RoboDK station: NewNozzleTest.rdk

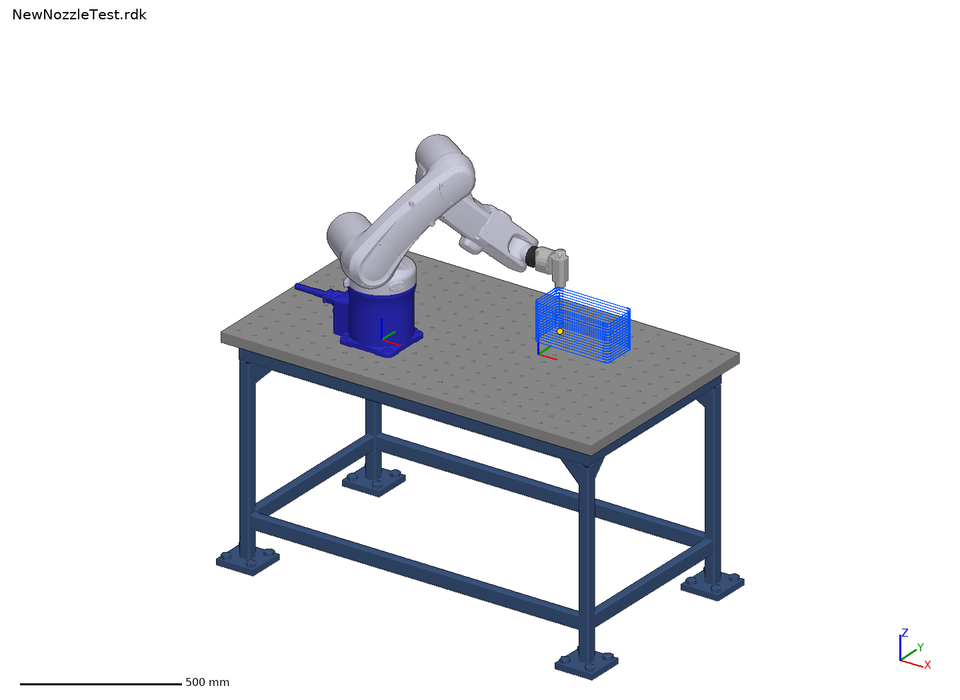
[picture v0: the station drawn from its stored meshes, robots at their saved joint values, targets as dots, program paths as lines]
Station NewNozzleTest (saved by RoboDK 5.5.4). Poses are relative to the parent item; angles as X-Y-Z fixed-axis rotations.
Station parameters (name, value as stored): TAGS, ['Additive Manufacturing', 'Additive manufacturing']
  - frame Denso VS-6577G-B Base at (0, 0, 0) mm
    - robot Denso VS-6577G-B: 6 axes, payload 7 kg, reach 854 mm, repeatability 0.03 mm, weight 36 kg
        modified DH rows (alpha deg, a mm, theta deg, d mm): 0, 0, 0, 335; -90, 75, -90, 0; 0, 365, -90, 0; -90, 90, 0, 405; 90, 0, 0, 0; -90, 0, 0, 80
        joint limits [-170, -100, -119, -190, -120, -360] to [170, 135, 169, 190, 120, 360]; home [0, 0, 90, 0, 0, 0]; saved at [-126.274, -49.631, -82.283, 63.884, 63.879, -41.926]
      - tool nozzle, TCP at (80, 0, 80) mm, rotated rx 0 ry 90 rz 0 deg, size 127 x 69.8 x 103.1 mm, geometry from nozzle.STEP
      - tool nozzle, TCP at (0, 0, 200) mm, size 127 x 76.2 x 113.3 mm, geometry from nozzle.STEP
    - object Table 1400x800x800mm at (-100, 160, 0) mm, size 1420 x 820 x 800 mm, geometry from Table-1400x800x800mm.sld
  - frame Reference at (454.66, 194.92, 0) mm
    - object Part at (0, 0, -20) mm, size 120 x 120 x 160 mm, geometry from part.sld
  - machining project Print3D settings: C:/Users/silverBlacK/OneDrive - University of Idaho/Research/RoboticsResearch/WallSection.gcode | rotZ(0) | rotX(0)*rotY(0) | rotZ(0)
  - program Print3D (17607 instructions, listed below)
  - Python program Extruder (listed below)
  - Python program SimulateFinalResult (listed below)
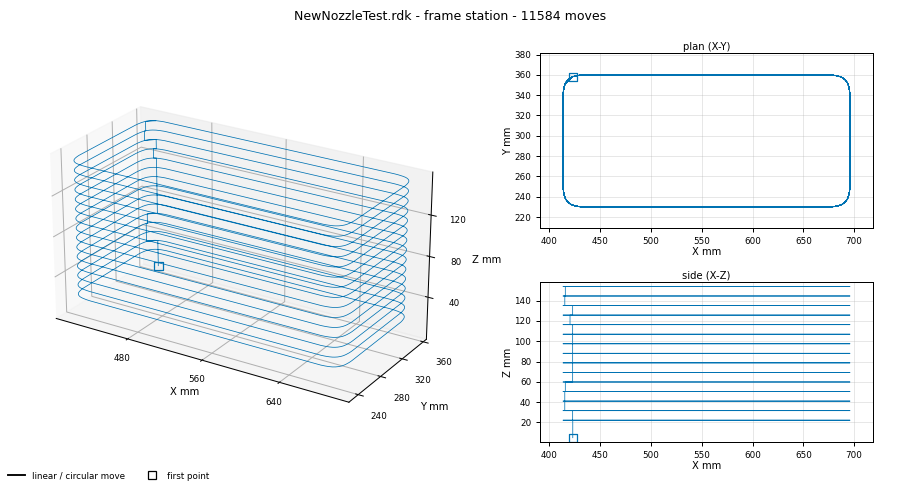
[picture p0: tool path of NewNozzleTest.rdk in frame station, 11584 of 11584 moves have a stored position in this frame; points joined in program order, loops and branches not executed]

--- program Print3D (robot Denso VS-6577G-B) ---
  Call M_RunCode(107)
  Call M_RunCode(104)
  Set speed (83.3 mm/s)
  Set speed (1000.0 mm/s)
  Set Ref.: Reference
  Set Tool: nozzle
  Show nozzle
  MoveJ 1 to (-31.64, 163.21, 5) mm, rotated rx -180 ry 0 rz 180 deg; joints [-126.294, -69.901, -72.383, 59.845, 68.77, -31.936]
  MoveL 2 to (-31.64, 163.21, 5) mm, rotated rx -180 ry 0 rz 180 deg; joints [-126.294, -69.901, -72.383, 59.845, 68.77, -31.936]
  Call Extruder(-1)
  MoveL 3 to (-31.64, 163.21, 5) mm, rotated rx -180 ry 0 rz 180 deg; joints [-126.294, -69.901, -72.383, 59.845, 68.77, -31.936]
  Call M_RunCode(109)
  Call M_RunCode(82)
  Call Extruder(0.00000)
  Set speed (130.0 mm/s)
  MoveL 4 to (-31.64, 163.21, 22.22) mm, rotated rx -180 ry 0 rz -180 deg; joints [-126.294, -67.456, -73.96, 60.14, 68.336, -32.743]
  Call Extruder(-2.00000)
  Set speed (40.0 mm/s)
  MoveL 5 to (-31.64, 163.21, 22.22) mm, rotated rx -180 ry 0 rz -180 deg; joints [-126.294, -67.456, -73.96, 60.14, 68.336, -32.743]
  Call Extruder(0.00000)
  Set speed (130.0 mm/s)
  MoveL 6 to (-31.64, 163.21, 22.22) mm, rotated rx -180 ry 0 rz -180 deg; joints [-126.294, -67.456, -73.96, 60.14, 68.336, -32.743]
  Call Extruder(2.00000)
  Set speed (40.0 mm/s)
  MoveL 7 to (-31.64, 163.21, 22.22) mm, rotated rx -180 ry 0 rz -180 deg; joints [-126.294, -67.456, -73.96, 60.14, 68.336, -32.743]
  Set speed (30.0 mm/s)
  MoveL 8 to (-31.64, 163.21, 22.22) mm, rotated rx -180 ry 0 rz -180 deg; joints [-126.294, -67.456, -73.96, 60.14, 68.336, -32.743]
  Call Extruder(2.38024)
  MoveL 9 to (-31.93, 163.09, 22.23) mm, rotated rx 180 ry 0 rz -180 deg; joints [-126.273, -67.437, -74.013, 60.147, 68.364, -32.718]
  MoveL 10 to (-31.93, 163.09, 22.23) mm, rotated rx 180 ry 0 rz -180 deg; joints [-126.273, -67.437, -74.013, 60.147, 68.364, -32.718]
  Call Extruder(2.76227)
  MoveL 11 to (-32.22, 162.97, 22.23) mm, rotated rx 180 ry 0 rz 180 deg; joints [-126.252, -67.418, -74.067, 60.155, 68.393, -32.692]
  MoveL 12 to (-32.22, 162.97, 22.23) mm, rotated rx 180 ry 0 rz 180 deg; joints [-126.252, -67.418, -74.067, 60.155, 68.393, -32.692]
  Call Extruder(3.11872)
  MoveL 13 to (-32.49, 162.85, 22.23) mm, rotated rx -180 ry 0 rz 180 deg; joints [-126.233, -67.401, -74.116, 60.161, 68.419, -32.669]
  MoveL 14 to (-32.49, 162.85, 22.23) mm, rotated rx -180 ry 0 rz 180 deg; joints [-126.233, -67.401, -74.116, 60.161, 68.419, -32.669]
  Call Extruder(3.44932)
  MoveL 15 to (-32.74, 162.74, 22.23) mm, rotated rx 180 ry 0 rz -180 deg; joints [-126.215, -67.385, -74.162, 60.167, 68.444, -32.647]
  MoveL 16 to (-32.74, 162.74, 22.23) mm, rotated rx 180 ry 0 rz -180 deg; joints [-126.215, -67.385, -74.162, 60.167, 68.444, -32.647]
  Call Extruder(3.78134)
  MoveL 17 to (-32.99, 162.64, 22.22) mm, rotated rx -180 ry 0 rz 180 deg; joints [-126.197, -67.369, -74.208, 60.173, 68.468, -32.625]
  MoveL 18 to (-32.99, 162.64, 22.22) mm, rotated rx -180 ry 0 rz 180 deg; joints [-126.197, -67.369, -74.208, 60.173, 68.468, -32.625]
  Call Extruder(4.21321)
  MoveL 19 to (-33.29, 162.46, 22.23) mm, rotated rx -180 ry 0 rz 180 deg; joints [-126.179, -67.347, -74.271, 60.176, 68.499, -32.593]
  MoveL 20 to (-33.29, 162.46, 22.23) mm, rotated rx -180 ry 0 rz 180 deg; joints [-126.179, -67.347, -74.271, 60.176, 68.499, -32.593]
  Call Extruder(4.64692)
  MoveL 21 to (-33.6, 162.29, 22.22) mm, rotated rx 180 ry 0 rz -180 deg; joints [-126.16, -67.325, -74.334, 60.178, 68.529, -32.561]
  MoveL 22 to (-33.6, 162.29, 22.22) mm, rotated rx 180 ry 0 rz -180 deg; joints [-126.16, -67.325, -74.334, 60.178, 68.529, -32.561]
  Call Extruder(5.08247)
  MoveL 23 to (-33.9, 162.11, 22.23) mm, rotated rx 180 ry 0 rz 180 deg; joints [-126.142, -67.303, -74.397, 60.181, 68.559, -32.529]
  MoveL 24 to (-33.9, 162.11, 22.23) mm, rotated rx 180 ry 0 rz 180 deg; joints [-126.142, -67.303, -74.397, 60.181, 68.559, -32.529]
  Call Extruder(5.51986)
  MoveL 25 to (-34.21, 161.94, 22.23) mm, rotated rx 180 ry 0 rz 180 deg; joints [-126.123, -67.281, -74.46, 60.184, 68.589, -32.497]
  MoveL 26 to (-34.21, 161.94, 22.23) mm, rotated rx 180 ry 0 rz 180 deg; joints [-126.123, -67.281, -74.46, 60.184, 68.589, -32.497]
  Call Extruder(5.89660)
  MoveL 27 to (-34.45, 161.76, 22.23) mm, rotated rx 180 ry 0 rz 180 deg; joints [-126.111, -67.261, -74.516, 60.182, 68.614, -32.467]
  MoveL 28 to (-34.45, 161.76, 22.23) mm, rotated rx 180 ry 0 rz 180 deg; joints [-126.111, -67.261, -74.516, 60.182, 68.614, -32.467]
  Call Extruder(6.59657)
  MoveL 29 to (-34.9, 161.43, 22.23) mm, rotated rx -180 ry 0 rz 180 deg; joints [-126.089, -67.225, -74.62, 60.18, 68.66, -32.411]
  MoveL 30 to (-34.9, 161.43, 22.23) mm, rotated rx -180 ry 0 rz 180 deg; joints [-126.089, -67.225, -74.62, 60.18, 68.66, -32.411]
  Call Extruder(7.29934)
  MoveL 31 to (-35.35, 161.1, 22.22) mm, rotated rx 180 ry 0 rz 180 deg; joints [-126.067, -67.189, -74.723, 60.177, 68.705, -32.355]
  Call Extruder(9.03811)
  MoveL 32 to (-36.39, 160.19, 22.22) mm, rotated rx 180 ry 0 rz 180 deg; joints [-126.027, -67.098, -74.986, 60.155, 68.812, -32.208]
  Call Extruder(10.77694)
  MoveL 33 to (-37.3, 159.15, 22.22) mm, rotated rx 180 ry 0 rz -180 deg; joints [-126.011, -67.006, -75.254, 60.111, 68.908, -32.051]
  Call Extruder(11.12832)
  MoveL 34 to (-37.47, 158.93, 22.22) mm, rotated rx -180 ry 0 rz 180 deg; joints [-126.011, -66.987, -75.308, 60.099, 68.926, -32.018]
  MoveL 35 to (-37.47, 158.93, 22.22) mm, rotated rx -180 ry 0 rz 180 deg; joints [-126.011, -66.987, -75.308, 60.099, 68.926, -32.018]
  Call Extruder(11.82828)
  MoveL 36 to (-37.79, 158.48, 22.22) mm, rotated rx 180 ry 0 rz 180 deg; joints [-126.011, -66.95, -75.416, 60.076, 68.961, -31.952]
  MoveL 37 to (-37.79, 158.48, 22.22) mm, rotated rx 180 ry 0 rz 180 deg; joints [-126.011, -66.95, -75.416, 60.076, 68.961, -31.952]
  Call Extruder(12.52544)
  MoveL 38 to (-38.12, 158.03, 22.23) mm, rotated rx 180 ry 0 rz 180 deg; joints [-126.011, -66.913, -75.524, 60.052, 68.996, -31.886]
  MoveL 39 to (-38.12, 158.03, 22.23) mm, rotated rx 180 ry 0 rz 180 deg; joints [-126.011, -66.913, -75.524, 60.052, 68.996, -31.886]
  Call Extruder(12.77229)
  MoveL 40 to (-38.22, 157.85, 22.23) mm, rotated rx 180 ry 0 rz -180 deg; joints [-126.013, -66.9, -75.562, 60.041, 69.008, -31.862]
  MoveL 41 to (-38.22, 157.85, 22.23) mm, rotated rx 180 ry 0 rz -180 deg; joints [-126.013, -66.9, -75.562, 60.041, 69.008, -31.862]
  Call Extruder(13.20785)
  MoveL 42 to (-38.4, 157.55, 22.22) mm, rotated rx -180 ry 0 rz -180 deg; joints [-126.018, -66.876, -75.63, 60.022, 69.027, -31.82]
  MoveL 43 to (-38.4, 157.55, 22.22) mm, rotated rx -180 ry 0 rz -180 deg; joints [-126.018, -66.876, -75.63, 60.022, 69.027, -31.82]
  Call Extruder(13.64157)
  MoveL 44 to (-38.57, 157.25, 22.22) mm, rotated rx 180 ry 0 rz -180 deg; joints [-126.023, -66.853, -75.697, 60.003, 69.047, -31.777]
  MoveL 45 to (-38.57, 157.25, 22.22) mm, rotated rx 180 ry 0 rz -180 deg; joints [-126.023, -66.853, -75.697, 60.003, 69.047, -31.777]
  Call Extruder(14.07344)
  MoveL 46 to (-38.75, 156.94, 22.22) mm, rotated rx -180 ry 0 rz -180 deg; joints [-126.028, -66.83, -75.765, 59.984, 69.066, -31.734]
  MoveL 47 to (-38.75, 156.94, 22.22) mm, rotated rx -180 ry 0 rz -180 deg; joints [-126.028, -66.83, -75.765, 59.984, 69.066, -31.734]
  Call Extruder(14.45383)
  MoveL 48 to (-38.89, 156.67, 22.22) mm, rotated rx -180 ry 0 rz -180 deg; joints [-126.034, -66.81, -75.824, 59.965, 69.083, -31.696]
  MoveL 49 to (-38.89, 156.67, 22.22) mm, rotated rx -180 ry 0 rz -180 deg; joints [-126.034, -66.81, -75.824, 59.965, 69.083, -31.696]
  Call Extruder(14.78446)
  MoveL 50 to (-39, 156.42, 22.22) mm, rotated rx -180 ry 0 rz -180 deg; joints [-126.042, -66.793, -75.875, 59.947, 69.095, -31.662]
  MoveL 51 to (-39, 156.42, 22.22) mm, rotated rx -180 ry 0 rz -180 deg; joints [-126.042, -66.793, -75.875, 59.947, 69.095, -31.662]
  Call Extruder(15.11366)
  MoveL 52 to (-39.1, 156.17, 22.23) mm, rotated rx -180 ry 0 rz 180 deg; joints [-126.05, -66.775, -75.926, 59.929, 69.108, -31.629]
  MoveL 53 to (-39.1, 156.17, 22.23) mm, rotated rx -180 ry 0 rz 180 deg; joints [-126.05, -66.775, -75.926, 59.929, 69.108, -31.629]
  Call Extruder(15.49565)
  MoveL 54 to (-39.23, 155.87, 22.22) mm, rotated rx -180 ry 0 rz -180 deg; joints [-126.06, -66.755, -75.985, 59.907, 69.122, -31.589]
  MoveL 55 to (-39.23, 155.87, 22.22) mm, rotated rx -180 ry 0 rz -180 deg; joints [-126.06, -66.755, -75.985, 59.907, 69.122, -31.589]
  Call Extruder(15.87585)
  MoveL 56 to (-39.35, 155.58, 22.22) mm, rotated rx -180 ry 0 rz 180 deg; joints [-126.07, -66.735, -76.044, 59.885, 69.137, -31.55]
  MoveL 57 to (-39.35, 155.58, 22.22) mm, rotated rx -180 ry 0 rz 180 deg; joints [-126.07, -66.735, -76.044, 59.885, 69.137, -31.55]
  Call Extruder(16.18353)
  MoveL 58 to (-39.44, 155.34, 22.22) mm, rotated rx 180 ry 0 rz -180 deg; joints [-126.079, -66.719, -76.092, 59.866, 69.148, -31.518]
  MoveL 59 to (-39.44, 155.34, 22.22) mm, rotated rx 180 ry 0 rz -180 deg; joints [-126.079, -66.719, -76.092, 59.866, 69.148, -31.518]
  Call Extruder(16.41988)
  MoveL 60 to (-39.5, 155.15, 22.22) mm, rotated rx -180 ry 0 rz 180 deg; joints [-126.087, -66.706, -76.128, 59.851, 69.156, -31.493]
  MoveL 61 to (-39.5, 155.15, 22.22) mm, rotated rx -180 ry 0 rz 180 deg; joints [-126.087, -66.706, -76.128, 59.851, 69.156, -31.493]
  Call Extruder(16.65518)
  MoveL 62 to (-39.56, 154.97, 22.23) mm, rotated rx 180 ry 0 rz -180 deg; joints [-126.095, -66.694, -76.164, 59.836, 69.163, -31.468]
  MoveL 63 to (-39.56, 154.97, 22.23) mm, rotated rx 180 ry 0 rz -180 deg; joints [-126.095, -66.694, -76.164, 59.836, 69.163, -31.468]
  Call Extruder(16.88943)
  MoveL 64 to (-39.62, 154.78, 22.22) mm, rotated rx -180 ry 0 rz -180 deg; joints [-126.103, -66.682, -76.201, 59.82, 69.171, -31.444]
  MoveL 65 to (-39.62, 154.78, 22.22) mm, rotated rx -180 ry 0 rz -180 deg; joints [-126.103, -66.682, -76.201, 59.82, 69.171, -31.444]
  Call Extruder(17.12262)
  MoveL 66 to (-39.68, 154.59, 22.22) mm, rotated rx 180 ry 0 rz 180 deg; joints [-126.111, -66.669, -76.237, 59.805, 69.179, -31.419]
  MoveL 67 to (-39.68, 154.59, 22.22) mm, rotated rx 180 ry 0 rz 180 deg; joints [-126.111, -66.669, -76.237, 59.805, 69.179, -31.419]
  Call Extruder(17.37548)
  MoveL 68 to (-39.75, 154.38, 22.22) mm, rotated rx 180 ry 0 rz 180 deg; joints [-126.12, -66.656, -76.276, 59.788, 69.187, -31.392]
  MoveL 69 to (-39.75, 154.38, 22.22) mm, rotated rx 180 ry 0 rz 180 deg; joints [-126.12, -66.656, -76.276, 59.788, 69.187, -31.392]
  Call Extruder(17.64775)
  MoveL 70 to (-39.81, 154.16, 22.23) mm, rotated rx 180 ry 0 rz 180 deg; joints [-126.131, -66.642, -76.318, 59.77, 69.196, -31.363]
  MoveL 71 to (-39.81, 154.16, 22.23) mm, rotated rx 180 ry 0 rz 180 deg; joints [-126.131, -66.642, -76.318, 59.77, 69.196, -31.363]
  Call Extruder(17.91868)
  MoveL 72 to (-39.88, 153.94, 22.23) mm, rotated rx -180 ry 0 rz 180 deg; joints [-126.141, -66.627, -76.361, 59.751, 69.205, -31.334]
  MoveL 73 to (-39.88, 153.94, 22.23) mm, rotated rx -180 ry 0 rz 180 deg; joints [-126.141, -66.627, -76.361, 59.751, 69.205, -31.334]
  Call Extruder(18.18828)
  MoveL 74 to (-39.95, 153.71, 22.23) mm, rotated rx 180 ry 0 rz -180 deg; joints [-126.151, -66.613, -76.403, 59.733, 69.213, -31.305]
  MoveL 75 to (-39.95, 153.71, 22.23) mm, rotated rx 180 ry 0 rz -180 deg; joints [-126.151, -66.613, -76.403, 59.733, 69.213, -31.305]
  Call Extruder(18.45654)
  MoveL 76 to (-40.02, 153.49, 22.22) mm, rotated rx -180 ry 0 rz 180 deg; joints [-126.161, -66.599, -76.445, 59.714, 69.222, -31.275]
  MoveL 77 to (-40.02, 153.49, 22.22) mm, rotated rx -180 ry 0 rz 180 deg; joints [-126.161, -66.599, -76.445, 59.714, 69.222, -31.275]
  Call Extruder(18.69554)
  MoveL 78 to (-40.06, 153.28, 22.23) mm, rotated rx 180 ry 0 rz 180 deg; joints [-126.173, -66.586, -76.482, 59.696, 69.228, -31.249]
  MoveL 79 to (-40.06, 153.28, 22.23) mm, rotated rx 180 ry 0 rz 180 deg; joints [-126.173, -66.586, -76.482, 59.696, 69.228, -31.249]
  Call Extruder(18.93348)
  MoveL 80 to (-40.11, 153.08, 22.23) mm, rotated rx 180 ry 0 rz 180 deg; joints [-126.184, -66.574, -76.518, 59.678, 69.235, -31.223]
  MoveL 81 to (-40.11, 153.08, 22.23) mm, rotated rx 180 ry 0 rz 180 deg; joints [-126.184, -66.574, -76.518, 59.678, 69.235, -31.223]
  Call Extruder(19.17035)
  MoveL 82 to (-40.15, 152.88, 22.22) mm, rotated rx 180 ry 0 rz 180 deg; joints [-126.195, -66.561, -76.555, 59.66, 69.241, -31.197]
  MoveL 83 to (-40.15, 152.88, 22.22) mm, rotated rx 180 ry 0 rz 180 deg; joints [-126.195, -66.561, -76.555, 59.66, 69.241, -31.197]
  Call Extruder(19.40615)
  MoveL 84 to (-40.2, 152.67, 22.22) mm, rotated rx -180 ry 0 rz 180 deg; joints [-126.206, -66.549, -76.592, 59.641, 69.248, -31.171]
  MoveL 85 to (-40.2, 152.67, 22.22) mm, rotated rx -180 ry 0 rz 180 deg; joints [-126.206, -66.549, -76.592, 59.641, 69.248, -31.171]
  Call Extruder(19.66605)
  MoveL 86 to (-40.24, 152.45, 22.23) mm, rotated rx 180 ry 0 rz 180 deg; joints [-126.219, -66.535, -76.632, 59.621, 69.255, -31.143]
  MoveL 87 to (-40.24, 152.45, 22.23) mm, rotated rx 180 ry 0 rz 180 deg; joints [-126.219, -66.535, -76.632, 59.621, 69.255, -31.143]
  Call Extruder(19.94972)
  MoveL 88 to (-40.29, 152.2, 22.22) mm, rotated rx 180 ry 0 rz -180 deg; joints [-126.233, -66.521, -76.676, 59.598, 69.262, -31.111]
  MoveL 89 to (-40.29, 152.2, 22.22) mm, rotated rx 180 ry 0 rz -180 deg; joints [-126.233, -66.521, -76.676, 59.598, 69.262, -31.111]
  Call Extruder(20.23193)
  MoveL 90 to (-40.34, 151.95, 22.22) mm, rotated rx -180 ry 0 rz 180 deg; joints [-126.248, -66.506, -76.72, 59.576, 69.269, -31.079]
  MoveL 91 to (-40.34, 151.95, 22.22) mm, rotated rx -180 ry 0 rz 180 deg; joints [-126.248, -66.506, -76.72, 59.576, 69.269, -31.079]
  Call Extruder(20.51271)
  MoveL 92 to (-40.39, 151.7, 22.23) mm, rotated rx 180 ry 0 rz 180 deg; joints [-126.262, -66.491, -76.764, 59.553, 69.277, -31.048]
  MoveL 93 to (-40.39, 151.7, 22.23) mm, rotated rx 180 ry 0 rz 180 deg; joints [-126.262, -66.491, -76.764, 59.553, 69.277, -31.048]
  Call Extruder(20.79205)
  MoveL 94 to (-40.44, 151.45, 22.22) mm, rotated rx -180 ry 0 rz 180 deg; joints [-126.276, -66.476, -76.808, 59.53, 69.284, -31.016]
  MoveL 95 to (-40.44, 151.45, 22.22) mm, rotated rx -180 ry 0 rz 180 deg; joints [-126.276, -66.476, -76.808, 59.53, 69.284, -31.016]
  Call Extruder(21.06994)
  MoveL 96 to (-40.49, 151.2, 22.23) mm, rotated rx 180 ry 0 rz 180 deg; joints [-126.291, -66.461, -76.852, 59.508, 69.292, -30.985]
  MoveL 97 to (-40.49, 151.2, 22.23) mm, rotated rx 180 ry 0 rz 180 deg; joints [-126.291, -66.461, -76.852, 59.508, 69.292, -30.985]
  Call Extruder(21.34639)
  MoveL 98 to (-40.54, 150.95, 22.22) mm, rotated rx -180 ry 0 rz -180 deg; joints [-126.305, -66.447, -76.896, 59.485, 69.299, -30.953]
  MoveL 99 to (-40.54, 150.95, 22.22) mm, rotated rx -180 ry 0 rz -180 deg; joints [-126.305, -66.447, -76.896, 59.485, 69.299, -30.953]
  Call Extruder(21.65140)
  MoveL 100 to (-40.59, 150.67, 22.22) mm, rotated rx 180 ry 0 rz 180 deg; joints [-126.322, -66.43, -76.944, 59.46, 69.307, -30.919]
  MoveL 101 to (-40.59, 150.67, 22.22) mm, rotated rx 180 ry 0 rz 180 deg; joints [-126.322, -66.43, -76.944, 59.46, 69.307, -30.919]
  Call Extruder(21.98479)
  MoveL 102 to (-40.64, 150.37, 22.22) mm, rotated rx -180 ry 0 rz 180 deg; joints [-126.341, -66.413, -76.996, 59.431, 69.315, -30.88]
  MoveL 103 to (-40.64, 150.37, 22.22) mm, rotated rx -180 ry 0 rz 180 deg; joints [-126.341, -66.413, -76.996, 59.431, 69.315, -30.88]
  Call Extruder(22.31647)
  MoveL 104 to (-40.69, 150.06, 22.23) mm, rotated rx -180 ry 0 rz 180 deg; joints [-126.36, -66.395, -77.049, 59.402, 69.322, -30.842]
  MoveL 105 to (-40.69, 150.06, 22.23) mm, rotated rx -180 ry 0 rz 180 deg; joints [-126.36, -66.395, -77.049, 59.402, 69.322, -30.842]
  Call Extruder(22.64643)
  MoveL 106 to (-40.74, 149.76, 22.22) mm, rotated rx -180 ry 0 rz -180 deg; joints [-126.379, -66.378, -77.101, 59.373, 69.33, -30.804]
  MoveL 107 to (-40.74, 149.76, 22.22) mm, rotated rx -180 ry 0 rz -180 deg; joints [-126.379, -66.378, -77.101, 59.373, 69.33, -30.804]
  Call Extruder(22.97467)
  MoveL 108 to (-40.78, 149.45, 22.22) mm, rotated rx -180 ry 0 rz -180 deg; joints [-126.398, -66.36, -77.153, 59.344, 69.338, -30.766]
  MoveL 109 to (-40.78, 149.45, 22.22) mm, rotated rx -180 ry 0 rz -180 deg; joints [-126.398, -66.36, -77.153, 59.344, 69.338, -30.766]
  Call Extruder(23.30119)
  MoveL 110 to (-40.83, 149.14, 22.22) mm, rotated rx 180 ry 0 rz -180 deg; joints [-126.417, -66.343, -77.206, 59.316, 69.346, -30.728]
  MoveL 111 to (-40.83, 149.14, 22.22) mm, rotated rx 180 ry 0 rz -180 deg; joints [-126.417, -66.343, -77.206, 59.316, 69.346, -30.728]
  Call Extruder(23.66827)
  MoveL 112 to (-40.88, 148.8, 22.22) mm, rotated rx 180 ry 0 rz -180 deg; joints [-126.439, -66.323, -77.264, 59.282, 69.355, -30.685]
  MoveL 113 to (-40.88, 148.8, 22.22) mm, rotated rx 180 ry 0 rz -180 deg; joints [-126.439, -66.323, -77.264, 59.282, 69.355, -30.685]
  Call Extruder(24.07571)
  MoveL 114 to (-40.92, 148.41, 22.22) mm, rotated rx -180 ry 0 rz 180 deg; joints [-126.465, -66.301, -77.328, 59.245, 69.363, -30.637]
  MoveL 115 to (-40.92, 148.41, 22.22) mm, rotated rx -180 ry 0 rz 180 deg; joints [-126.465, -66.301, -77.328, 59.245, 69.363, -30.637]
  Call Extruder(24.48110)
  MoveL 116 to (-40.97, 148.02, 22.22) mm, rotated rx -180 ry 0 rz -180 deg; joints [-126.491, -66.28, -77.393, 59.207, 69.372, -30.589]
  MoveL 117 to (-40.97, 148.02, 22.22) mm, rotated rx -180 ry 0 rz -180 deg; joints [-126.491, -66.28, -77.393, 59.207, 69.372, -30.589]
  Call Extruder(24.88445)
  MoveL 118 to (-41.02, 147.63, 22.23) mm, rotated rx 180 ry 0 rz -180 deg; joints [-126.517, -66.259, -77.457, 59.169, 69.381, -30.542]
  MoveL 119 to (-41.02, 147.63, 22.23) mm, rotated rx 180 ry 0 rz -180 deg; joints [-126.517, -66.259, -77.457, 59.169, 69.381, -30.542]
  Call Extruder(25.28574)
  MoveL 120 to (-41.06, 147.25, 22.22) mm, rotated rx -180 ry 0 rz 180 deg; joints [-126.543, -66.237, -77.521, 59.131, 69.389, -30.494]
  MoveL 121 to (-41.06, 147.25, 22.22) mm, rotated rx -180 ry 0 rz 180 deg; joints [-126.543, -66.237, -77.521, 59.131, 69.389, -30.494]
  Call Extruder(25.89062)
  MoveL 122 to (-41.11, 146.66, 22.23) mm, rotated rx -180 ry 0 rz 180 deg; joints [-126.585, -66.206, -77.616, 59.072, 69.401, -30.422]
  MoveL 123 to (-41.11, 146.66, 22.23) mm, rotated rx -180 ry 0 rz 180 deg; joints [-126.585, -66.206, -77.616, 59.072, 69.401, -30.422]
  Call Extruder(26.49235)
  MoveL 124 to (-41.15, 146.07, 22.23) mm, rotated rx 180 ry 0 rz -180 deg; joints [-126.628, -66.174, -77.711, 59.013, 69.412, -30.35]
  MoveL 125 to (-41.15, 146.07, 22.23) mm, rotated rx 180 ry 0 rz -180 deg; joints [-126.628, -66.174, -77.711, 59.013, 69.412, -30.35]
  Call Extruder(27.09093)
  MoveL 126 to (-41.2, 145.48, 22.23) mm, rotated rx -180 ry 0 rz 180 deg; joints [-126.67, -66.143, -77.806, 58.953, 69.423, -30.279]
  MoveL 127 to (-41.2, 145.48, 22.23) mm, rotated rx -180 ry 0 rz 180 deg; joints [-126.67, -66.143, -77.806, 58.953, 69.423, -30.279]
  Call Extruder(28.26271)
  MoveL 128 to (-41.25, 144.32, 22.23) mm, rotated rx 180 ry 0 rz 180 deg; joints [-126.759, -66.083, -77.987, 58.832, 69.441, -30.139]
  MoveL 129 to (-41.25, 144.32, 22.23) mm, rotated rx 180 ry 0 rz 180 deg; joints [-126.759, -66.083, -77.987, 58.832, 69.441, -30.139]
  Call Extruder(29.72057)
  MoveL 130 to (-41.29, 142.86, 22.23) mm, rotated rx 180 ry 0 rz 180 deg; joints [-126.873, -66.009, -78.211, 58.679, 69.462, -29.965]
  Call Extruder(115.61408)
  MoveL 131 to (-41.29, 57.14, 22.22) mm, rotated rx 180 ry 0 rz 180 deg; joints [-135.148, -62.641, -89.71, 48.318, 70.793, -20.278]
  Call Extruder(116.48916)
  MoveL 132 to (-41.27, 56.26, 22.23) mm, rotated rx 180 ry 0 rz 180 deg; joints [-135.25, -62.616, -89.811, 48.198, 70.808, -20.185]
  MoveL 133 to (-41.27, 56.26, 22.23) mm, rotated rx 180 ry 0 rz 180 deg; joints [-135.25, -62.616, -89.811, 48.198, 70.808, -20.185]
  Call Extruder(117.66094)
  MoveL 134 to (-41.23, 55.1, 22.22) mm, rotated rx -180 ry 0 rz 180 deg; joints [-135.387, -62.583, -89.942, 48.035, 70.826, -20.063]
  MoveL 135 to (-41.23, 55.1, 22.22) mm, rotated rx -180 ry 0 rz 180 deg; joints [-135.387, -62.583, -89.942, 48.035, 70.826, -20.063]
  Call Extruder(118.54904)
  MoveL 136 to (-41.18, 54.23, 22.23) mm, rotated rx 180 ry 0 rz 180 deg; joints [-135.493, -62.559, -90.039, 47.911, 70.839, -19.971]
  MoveL 137 to (-41.18, 54.23, 22.23) mm, rotated rx 180 ry 0 rz 180 deg; joints [-135.493, -62.559, -90.039, 47.911, 70.839, -19.971]
  Call Extruder(119.15077)
  MoveL 138 to (-41.13, 53.64, 22.23) mm, rotated rx 180 ry 0 rz 180 deg; joints [-135.566, -62.543, -90.102, 47.826, 70.846, -19.909]
  MoveL 139 to (-41.13, 53.64, 22.23) mm, rotated rx 180 ry 0 rz 180 deg; joints [-135.566, -62.543, -90.102, 47.826, 70.846, -19.909]
  Call Extruder(119.75565)
  MoveL 140 to (-41.09, 53.05, 22.22) mm, rotated rx -180 ry 0 rz -180 deg; joints [-135.64, -62.528, -90.165, 47.741, 70.853, -19.848]
  MoveL 141 to (-41.09, 53.05, 22.22) mm, rotated rx -180 ry 0 rz -180 deg; joints [-135.64, -62.528, -90.165, 47.741, 70.853, -19.848]
  Call Extruder(120.26021)
  MoveL 142 to (-41.04, 52.56, 22.23) mm, rotated rx 180 ry 0 rz 180 deg; joints [-135.701, -62.515, -90.217, 47.67, 70.858, -19.798]
  MoveL 143 to (-41.04, 52.56, 22.23) mm, rotated rx 180 ry 0 rz 180 deg; joints [-135.701, -62.515, -90.217, 47.67, 70.858, -19.798]
  Call Extruder(120.66355)
  MoveL 144 to (-40.99, 52.17, 22.23) mm, rotated rx -180 ry 0 rz 180 deg; joints [-135.751, -62.505, -90.256, 47.612, 70.862, -19.758]
  MoveL 145 to (-40.99, 52.17, 22.23) mm, rotated rx -180 ry 0 rz 180 deg; joints [-135.751, -62.505, -90.256, 47.612, 70.862, -19.758]
  Call Extruder(121.06894)
  MoveL 146 to (-40.95, 51.78, 22.23) mm, rotated rx 180 ry 0 rz 180 deg; joints [-135.801, -62.496, -90.296, 47.554, 70.865, -19.718]
  MoveL 147 to (-40.95, 51.78, 22.23) mm, rotated rx 180 ry 0 rz 180 deg; joints [-135.801, -62.496, -90.296, 47.554, 70.865, -19.718]
  Call Extruder(121.47639)
  MoveL 148 to (-40.9, 51.4, 22.23) mm, rotated rx 180 ry 0 rz -180 deg; joints [-135.852, -62.486, -90.335, 47.497, 70.868, -19.679]
  MoveL 149 to (-40.9, 51.4, 22.23) mm, rotated rx 180 ry 0 rz -180 deg; joints [-135.852, -62.486, -90.335, 47.497, 70.868, -19.679]
  Call Extruder(121.88588)
  MoveL 150 to (-40.86, 51.01, 22.23) mm, rotated rx 180 ry 0 rz 180 deg; joints [-135.902, -62.476, -90.375, 47.439, 70.871, -19.639]
  MoveL 151 to (-40.86, 51.01, 22.23) mm, rotated rx 180 ry 0 rz 180 deg; joints [-135.902, -62.476, -90.375, 47.439, 70.871, -19.639]
  Call Extruder(122.21240)
  MoveL 152 to (-40.81, 50.7, 22.23) mm, rotated rx 180 ry 0 rz -180 deg; joints [-135.943, -62.469, -90.404, 47.392, 70.873, -19.608]
  MoveL 153 to (-40.81, 50.7, 22.23) mm, rotated rx 180 ry 0 rz -180 deg; joints [-135.943, -62.469, -90.404, 47.392, 70.873, -19.608]
  Call Extruder(122.54064)
  MoveL 154 to (-40.76, 50.4, 22.22) mm, rotated rx 180 ry 0 rz -180 deg; joints [-135.984, -62.462, -90.434, 47.346, 70.874, -19.577]
  MoveL 155 to (-40.76, 50.4, 22.22) mm, rotated rx 180 ry 0 rz -180 deg; joints [-135.984, -62.462, -90.434, 47.346, 70.874, -19.577]
  Call Extruder(122.87060)
  MoveL 156 to (-40.71, 50.09, 22.23) mm, rotated rx 180 ry 0 rz 180 deg; joints [-136.025, -62.455, -90.463, 47.299, 70.875, -19.547]
  MoveL 157 to (-40.71, 50.09, 22.23) mm, rotated rx 180 ry 0 rz 180 deg; joints [-136.025, -62.455, -90.463, 47.299, 70.875, -19.547]
  Call Extruder(123.20228)
  MoveL 158 to (-40.66, 49.79, 22.23) mm, rotated rx 180 ry 0 rz -180 deg; joints [-136.067, -62.448, -90.493, 47.252, 70.876, -19.516]
  MoveL 159 to (-40.66, 49.79, 22.23) mm, rotated rx 180 ry 0 rz -180 deg; joints [-136.067, -62.448, -90.493, 47.252, 70.876, -19.516]
  Call Extruder(123.53568)
  MoveL 160 to (-40.61, 49.48, 22.23) mm, rotated rx 180 ry 0 rz 180 deg; joints [-136.108, -62.441, -90.522, 47.205, 70.878, -19.485]
  MoveL 161 to (-40.61, 49.48, 22.23) mm, rotated rx 180 ry 0 rz 180 deg; joints [-136.108, -62.441, -90.522, 47.205, 70.878, -19.485]
  Call Extruder(123.87079)
  MoveL 162 to (-40.56, 49.18, 22.23) mm, rotated rx 180 ry 0 rz 180 deg; joints [-136.149, -62.433, -90.551, 47.159, 70.879, -19.454]
  MoveL 163 to (-40.56, 49.18, 22.23) mm, rotated rx 180 ry 0 rz 180 deg; joints [-136.149, -62.433, -90.551, 47.159, 70.879, -19.454]
  Call Extruder(124.14680)
  MoveL 164 to (-40.52, 48.93, 22.23) mm, rotated rx 180 ry 0 rz 180 deg; joints [-136.184, -62.428, -90.574, 47.12, 70.879, -19.43]
  MoveL 165 to (-40.52, 48.93, 22.23) mm, rotated rx 180 ry 0 rz 180 deg; joints [-136.184, -62.428, -90.574, 47.12, 70.879, -19.43]
  Call Extruder(124.42424)
  MoveL 166 to (-40.47, 48.68, 22.22) mm, rotated rx 180 ry 0 rz 180 deg; joints [-136.219, -62.422, -90.597, 47.08, 70.879, -19.405]
  MoveL 167 to (-40.47, 48.68, 22.22) mm, rotated rx 180 ry 0 rz 180 deg; joints [-136.219, -62.422, -90.597, 47.08, 70.879, -19.405]
  Call Extruder(124.70312)
  MoveL 168 to (-40.42, 48.43, 22.23) mm, rotated rx 180 ry 0 rz 180 deg; joints [-136.253, -62.417, -90.62, 47.041, 70.88, -19.38]
  MoveL 169 to (-40.42, 48.43, 22.23) mm, rotated rx 180 ry 0 rz 180 deg; joints [-136.253, -62.417, -90.62, 47.041, 70.88, -19.38]
  Call Extruder(124.98344)
  MoveL 170 to (-40.37, 48.18, 22.23) mm, rotated rx 180 ry 0 rz 180 deg; joints [-136.288, -62.411, -90.642, 47.002, 70.88, -19.356]
  MoveL 171 to (-40.37, 48.18, 22.23) mm, rotated rx 180 ry 0 rz 180 deg; joints [-136.288, -62.411, -90.642, 47.002, 70.88, -19.356]
  Call Extruder(125.26519)
  MoveL 172 to (-40.32, 47.93, 22.23) mm, rotated rx 180 ry 0 rz 180 deg; joints [-136.323, -62.406, -90.665, 46.963, 70.88, -19.331]
  MoveL 173 to (-40.32, 47.93, 22.23) mm, rotated rx 180 ry 0 rz 180 deg; joints [-136.323, -62.406, -90.665, 46.963, 70.88, -19.331]
  Call Extruder(125.54838)
  MoveL 174 to (-40.27, 47.68, 22.22) mm, rotated rx -180 ry 0 rz 180 deg; joints [-136.358, -62.401, -90.687, 46.924, 70.88, -19.306]
  MoveL 175 to (-40.27, 47.68, 22.22) mm, rotated rx -180 ry 0 rz 180 deg; joints [-136.358, -62.401, -90.687, 46.924, 70.88, -19.306]
  Call Extruder(125.76334)
  MoveL 176 to (-40.23, 47.49, 22.23) mm, rotated rx 180 ry 0 rz -180 deg; joints [-136.384, -62.396, -90.704, 46.894, 70.88, -19.288]
  MoveL 177 to (-40.23, 47.49, 22.23) mm, rotated rx 180 ry 0 rz -180 deg; joints [-136.384, -62.396, -90.704, 46.894, 70.88, -19.288]
  Call Extruder(125.95387)
  MoveL 178 to (-40.2, 47.33, 22.23) mm, rotated rx 180 ry 0 rz 180 deg; joints [-136.408, -62.393, -90.719, 46.868, 70.88, -19.271]
  MoveL 179 to (-40.2, 47.33, 22.23) mm, rotated rx 180 ry 0 rz 180 deg; joints [-136.408, -62.393, -90.719, 46.868, 70.88, -19.271]
  Call Extruder(126.19017)
  MoveL 180 to (-40.15, 47.12, 22.23) mm, rotated rx 180 ry 0 rz 180 deg; joints [-136.437, -62.389, -90.737, 46.835, 70.88, -19.251]
  MoveL 181 to (-40.15, 47.12, 22.23) mm, rotated rx 180 ry 0 rz 180 deg; joints [-136.437, -62.389, -90.737, 46.835, 70.88, -19.251]
  Call Extruder(126.42754)
  MoveL 182 to (-40.11, 46.92, 22.23) mm, rotated rx 180 ry 0 rz 180 deg; joints [-136.466, -62.384, -90.755, 46.803, 70.879, -19.231]
  MoveL 183 to (-40.11, 46.92, 22.23) mm, rotated rx 180 ry 0 rz 180 deg; joints [-136.466, -62.384, -90.755, 46.803, 70.879, -19.231]
  Call Extruder(126.66598)
  MoveL 184 to (-40.06, 46.72, 22.23) mm, rotated rx 180 ry 0 rz 180 deg; joints [-136.495, -62.38, -90.773, 46.77, 70.879, -19.211]
  MoveL 185 to (-40.06, 46.72, 22.23) mm, rotated rx 180 ry 0 rz 180 deg; joints [-136.495, -62.38, -90.773, 46.77, 70.879, -19.211]
  Call Extruder(126.90549)
  MoveL 186 to (-40.02, 46.51, 22.23) mm, rotated rx 180 ry 0 rz 180 deg; joints [-136.525, -62.376, -90.791, 46.738, 70.879, -19.191]
  MoveL 187 to (-40.02, 46.51, 22.23) mm, rotated rx 180 ry 0 rz 180 deg; joints [-136.525, -62.376, -90.791, 46.738, 70.879, -19.191]
  Call Extruder(127.17442)
  MoveL 188 to (-39.95, 46.29, 22.22) mm, rotated rx 180 ry 0 rz 180 deg; joints [-136.559, -62.371, -90.808, 46.7, 70.877, -19.17]
  MoveL 189 to (-39.95, 46.29, 22.22) mm, rotated rx 180 ry 0 rz 180 deg; joints [-136.559, -62.371, -90.808, 46.7, 70.877, -19.17]
  Call Extruder(127.44468)
  MoveL 190 to (-39.88, 46.06, 22.23) mm, rotated rx 180 ry 0 rz -180 deg; joints [-136.593, -62.367, -90.825, 46.663, 70.874, -19.149]
  MoveL 191 to (-39.88, 46.06, 22.23) mm, rotated rx 180 ry 0 rz -180 deg; joints [-136.593, -62.367, -90.825, 46.663, 70.874, -19.149]
  Call Extruder(127.71628)
  MoveL 192 to (-39.81, 45.84, 22.23) mm, rotated rx 180 ry 0 rz 180 deg; joints [-136.627, -62.363, -90.843, 46.625, 70.872, -19.127]
  MoveL 193 to (-39.81, 45.84, 22.23) mm, rotated rx 180 ry 0 rz 180 deg; joints [-136.627, -62.363, -90.843, 46.625, 70.872, -19.127]
  Call Extruder(127.98921)
  MoveL 194 to (-39.75, 45.62, 22.23) mm, rotated rx 180 ry 0 rz 180 deg; joints [-136.661, -62.359, -90.86, 46.588, 70.87, -19.106]
  MoveL 195 to (-39.75, 45.62, 22.23) mm, rotated rx 180 ry 0 rz 180 deg; joints [-136.661, -62.359, -90.86, 46.588, 70.87, -19.106]
  Call Extruder(128.24265)
  MoveL 196 to (-39.68, 45.41, 22.22) mm, rotated rx 180 ry 0 rz 180 deg; joints [-136.693, -62.355, -90.875, 46.553, 70.868, -19.086]
  MoveL 197 to (-39.68, 45.41, 22.22) mm, rotated rx 180 ry 0 rz 180 deg; joints [-136.693, -62.355, -90.875, 46.553, 70.868, -19.086]
  Call Extruder(128.47637)
  MoveL 198 to (-39.62, 45.22, 22.23) mm, rotated rx -180 ry 0 rz 180 deg; joints [-136.722, -62.352, -90.889, 46.521, 70.865, -19.069]
  MoveL 199 to (-39.62, 45.22, 22.23) mm, rotated rx -180 ry 0 rz 180 deg; joints [-136.722, -62.352, -90.889, 46.521, 70.865, -19.069]
  Call Extruder(128.71114)
  MoveL 200 to (-39.56, 45.03, 22.22) mm, rotated rx 180 ry 0 rz 180 deg; joints [-136.751, -62.348, -90.904, 46.489, 70.863, -19.051]
  MoveL 201 to (-39.56, 45.03, 22.22) mm, rotated rx 180 ry 0 rz 180 deg; joints [-136.751, -62.348, -90.904, 46.489, 70.863, -19.051]
  Call Extruder(128.94697)
  MoveL 202 to (-39.5, 44.85, 22.23) mm, rotated rx -180 ry 0 rz -180 deg; joints [-136.781, -62.345, -90.918, 46.457, 70.861, -19.033]
  MoveL 203 to (-39.5, 44.85, 22.23) mm, rotated rx -180 ry 0 rz -180 deg; joints [-136.781, -62.345, -90.918, 46.457, 70.861, -19.033]
  Call Extruder(129.18384)
  MoveL 204 to (-39.44, 44.66, 22.23) mm, rotated rx -180 ry 0 rz -180 deg; joints [-136.81, -62.342, -90.931, 46.425, 70.859, -19.015]
  MoveL 205 to (-39.44, 44.66, 22.23) mm, rotated rx -180 ry 0 rz -180 deg; joints [-136.81, -62.342, -90.931, 46.425, 70.859, -19.015]
  Call Extruder(129.49225)
  MoveL 206 to (-39.35, 44.42, 22.23) mm, rotated rx 180 ry 0 rz 180 deg; joints [-136.849, -62.338, -90.948, 46.383, 70.855, -18.993]
  MoveL 207 to (-39.35, 44.42, 22.23) mm, rotated rx 180 ry 0 rz 180 deg; joints [-136.849, -62.338, -90.948, 46.383, 70.855, -18.993]
  Call Extruder(129.87335)
  MoveL 208 to (-39.23, 44.12, 22.22) mm, rotated rx -180 ry 0 rz 180 deg; joints [-136.898, -62.334, -90.966, 46.331, 70.848, -18.967]
  MoveL 209 to (-39.23, 44.12, 22.22) mm, rotated rx -180 ry 0 rz 180 deg; joints [-136.898, -62.334, -90.966, 46.331, 70.848, -18.967]
  Call Extruder(130.25623)
  MoveL 210 to (-39.11, 43.83, 22.22) mm, rotated rx 180 ry 0 rz 180 deg; joints [-136.946, -62.329, -90.984, 46.279, 70.842, -18.94]
  MoveL 211 to (-39.11, 43.83, 22.22) mm, rotated rx 180 ry 0 rz 180 deg; joints [-136.946, -62.329, -90.984, 46.279, 70.842, -18.94]
  Call Extruder(130.58614)
  MoveL 212 to (-39, 43.58, 22.22) mm, rotated rx 180 ry 0 rz -180 deg; joints [-136.988, -62.325, -91, 46.234, 70.837, -18.917]
  MoveL 213 to (-39, 43.58, 22.22) mm, rotated rx 180 ry 0 rz -180 deg; joints [-136.988, -62.325, -91, 46.234, 70.837, -18.917]
  Call Extruder(130.91747)
  MoveL 214 to (-38.89, 43.34, 22.23) mm, rotated rx -180 ry 0 rz 180 deg; joints [-137.029, -62.322, -91.015, 46.189, 70.831, -18.895]
  MoveL 215 to (-38.89, 43.34, 22.23) mm, rotated rx -180 ry 0 rz 180 deg; joints [-137.029, -62.322, -91.015, 46.189, 70.831, -18.895]
  Call Extruder(131.29867)
  MoveL 216 to (-38.75, 43.06, 22.22) mm, rotated rx 180 ry 0 rz 180 deg; joints [-137.078, -62.318, -91.029, 46.138, 70.823, -18.87]
  MoveL 217 to (-38.75, 43.06, 22.22) mm, rotated rx 180 ry 0 rz 180 deg; joints [-137.078, -62.318, -91.029, 46.138, 70.823, -18.87]
  Call Extruder(131.73146)
  MoveL 218 to (-38.57, 42.75, 22.23) mm, rotated rx -180 ry 0 rz -180 deg; joints [-137.135, -62.315, -91.042, 46.079, 70.812, -18.844]
  MoveL 219 to (-38.57, 42.75, 22.23) mm, rotated rx -180 ry 0 rz -180 deg; joints [-137.135, -62.315, -91.042, 46.079, 70.812, -18.844]
  Call Extruder(132.16610)
  MoveL 220 to (-38.4, 42.45, 22.23) mm, rotated rx 180 ry 0 rz -180 deg; joints [-137.191, -62.312, -91.055, 46.02, 70.8, -18.818]
  MoveL 221 to (-38.4, 42.45, 22.23) mm, rotated rx 180 ry 0 rz -180 deg; joints [-137.191, -62.312, -91.055, 46.02, 70.8, -18.818]
  Call Extruder(132.60257)
  MoveL 222 to (-38.22, 42.15, 22.23) mm, rotated rx 180 ry 0 rz -180 deg; joints [-137.247, -62.309, -91.067, 45.961, 70.789, -18.793]
  MoveL 223 to (-38.22, 42.15, 22.23) mm, rotated rx 180 ry 0 rz -180 deg; joints [-137.247, -62.309, -91.067, 45.961, 70.789, -18.793]
  Call Extruder(132.84952)
  MoveL 224 to (-38.12, 41.98, 22.23) mm, rotated rx -180 ry 0 rz 180 deg; joints [-137.279, -62.308, -91.075, 45.928, 70.783, -18.778]
  MoveL 225 to (-38.12, 41.98, 22.23) mm, rotated rx -180 ry 0 rz 180 deg; joints [-137.279, -62.308, -91.075, 45.928, 70.783, -18.778]
  Call Extruder(133.54809)
  MoveL 226 to (-37.8, 41.52, 22.22) mm, rotated rx -180 ry 0 rz 180 deg; joints [-137.37, -62.305, -91.085, 45.835, 70.759, -18.742]
  MoveL 227 to (-37.8, 41.52, 22.22) mm, rotated rx -180 ry 0 rz 180 deg; joints [-137.37, -62.305, -91.085, 45.835, 70.759, -18.742]
  Call Extruder(134.24946)
  MoveL 228 to (-37.47, 41.07, 22.22) mm, rotated rx -180 ry 0 rz 180 deg; joints [-137.461, -62.303, -91.096, 45.742, 70.735, -18.706]
  MoveL 229 to (-37.47, 41.07, 22.22) mm, rotated rx -180 ry 0 rz 180 deg; joints [-137.461, -62.303, -91.096, 45.742, 70.735, -18.706]
  Call Extruder(134.60151)
  MoveL 230 to (-37.3, 40.85, 22.23) mm, rotated rx 180 ry 0 rz 180 deg; joints [-137.506, -62.301, -91.101, 45.695, 70.723, -18.687]
  Call Extruder(136.34360)
  MoveL 231 to (-36.39, 39.81, 22.23) mm, rotated rx 180 ry 0 rz -180 deg; joints [-137.733, -62.3, -91.105, 45.467, 70.653, -18.61]
  Call Extruder(137.66925)
  MoveL 232 to (-35.6, 39.11, 22.23) mm, rotated rx 180 ry 0 rz 180 deg; joints [-137.904, -62.305, -91.086, 45.298, 70.588, -18.563]
  MoveL 233 to (-35.6, 39.11, 22.23) mm, rotated rx 180 ry 0 rz 180 deg; joints [-137.904, -62.305, -91.086, 45.298, 70.588, -18.563]
  Call Extruder(138.08410)
  MoveL 234 to (-35.35, 38.9, 22.23) mm, rotated rx -180 ry 0 rz -180 deg; joints [-137.958, -62.306, -91.079, 45.245, 70.568, -18.549]
  Call Extruder(138.78545)
  MoveL 235 to (-34.9, 38.57, 22.23) mm, rotated rx 180 ry 0 rz -180 deg; joints [-138.048, -62.311, -91.06, 45.159, 70.529, -18.53]
  MoveL 236 to (-34.9, 38.57, 22.23) mm, rotated rx 180 ry 0 rz -180 deg; joints [-138.048, -62.311, -91.06, 45.159, 70.529, -18.53]
  Call Extruder(139.48400)
  MoveL 237 to (-34.45, 38.24, 22.23) mm, rotated rx 180 ry 0 rz 180 deg; joints [-138.137, -62.316, -91.041, 45.073, 70.49, -18.511]
  MoveL 238 to (-34.45, 38.24, 22.23) mm, rotated rx 180 ry 0 rz 180 deg; joints [-138.137, -62.316, -91.041, 45.073, 70.49, -18.511]
  Call Extruder(139.86003)
  MoveL 239 to (-34.21, 38.06, 22.23) mm, rotated rx -180 ry 0 rz 180 deg; joints [-138.185, -62.318, -91.03, 45.026, 70.469, -18.501]
  MoveL 240 to (-34.21, 38.06, 22.23) mm, rotated rx -180 ry 0 rz 180 deg; joints [-138.185, -62.318, -91.03, 45.026, 70.469, -18.501]
  Call Extruder(140.29650)
  MoveL 241 to (-33.9, 37.89, 22.23) mm, rotated rx 180 ry 0 rz -180 deg; joints [-138.24, -62.323, -91.012, 44.974, 70.442, -18.493]
  MoveL 242 to (-33.9, 37.89, 22.23) mm, rotated rx 180 ry 0 rz -180 deg; joints [-138.24, -62.323, -91.012, 44.974, 70.442, -18.493]
  Call Extruder(140.73113)
  MoveL 243 to (-33.6, 37.71, 22.23) mm, rotated rx 180 ry 0 rz 180 deg; joints [-138.295, -62.327, -90.994, 44.923, 70.415, -18.485]
  MoveL 244 to (-33.6, 37.71, 22.23) mm, rotated rx 180 ry 0 rz 180 deg; joints [-138.295, -62.327, -90.994, 44.923, 70.415, -18.485]
  Call Extruder(141.16391)
  MoveL 245 to (-33.29, 37.54, 22.23) mm, rotated rx -180 ry 0 rz 180 deg; joints [-138.349, -62.331, -90.976, 44.871, 70.388, -18.477]
  MoveL 246 to (-33.29, 37.54, 22.23) mm, rotated rx -180 ry 0 rz 180 deg; joints [-138.349, -62.331, -90.976, 44.871, 70.388, -18.477]
  Call Extruder(141.59485)
  MoveL 247 to (-32.99, 37.36, 22.23) mm, rotated rx 180 ry 0 rz 180 deg; joints [-138.404, -62.336, -90.957, 44.82, 70.36, -18.469]
  MoveL 248 to (-32.99, 37.36, 22.23) mm, rotated rx 180 ry 0 rz 180 deg; joints [-138.404, -62.336, -90.957, 44.82, 70.36, -18.469]
  Call Extruder(141.92621)
  MoveL 249 to (-32.74, 37.26, 22.22) mm, rotated rx -180 ry 0 rz -180 deg; joints [-138.444, -62.34, -90.938, 44.783, 70.337, -18.467]
  MoveL 250 to (-32.74, 37.26, 22.22) mm, rotated rx -180 ry 0 rz -180 deg; joints [-138.444, -62.34, -90.938, 44.783, 70.337, -18.467]
  Call Extruder(142.25615)
  MoveL 251 to (-32.49, 37.15, 22.23) mm, rotated rx 180 ry 0 rz 180 deg; joints [-138.484, -62.345, -90.919, 44.746, 70.314, -18.464]
  MoveL 252 to (-32.49, 37.15, 22.23) mm, rotated rx 180 ry 0 rz 180 deg; joints [-138.484, -62.345, -90.919, 44.746, 70.314, -18.464]
  Call Extruder(142.61184)
  MoveL 253 to (-32.22, 37.03, 22.22) mm, rotated rx -180 ry 0 rz 180 deg; joints [-138.527, -62.35, -90.898, 44.707, 70.289, -18.461]
  MoveL 254 to (-32.22, 37.03, 22.22) mm, rotated rx -180 ry 0 rz 180 deg; joints [-138.527, -62.35, -90.898, 44.707, 70.289, -18.461]
  Call Extruder(142.99292)
  MoveL 255 to (-31.93, 36.91, 22.23) mm, rotated rx -180 ry 0 rz 180 deg; joints [-138.574, -62.355, -90.875, 44.664, 70.262, -18.458]
  MoveL 256 to (-31.93, 36.91, 22.23) mm, rotated rx -180 ry 0 rz 180 deg; joints [-138.574, -62.355, -90.875, 44.664, 70.262, -18.458]
  Call Extruder(143.37221)
  MoveL 257 to (-31.64, 36.79, 22.22) mm, rotated rx 180 ry 0 rz 180 deg; joints [-138.62, -62.361, -90.852, 44.622, 70.235, -18.455]
  MoveL 258 to (-31.64, 36.79, 22.22) mm, rotated rx 180 ry 0 rz 180 deg; joints [-138.62, -62.361, -90.852, 44.622, 70.235, -18.455]
  Call Extruder(143.60909)
  MoveL 259 to (-31.45, 36.73, 22.23) mm, rotated rx -180 ry 0 rz 180 deg; joints [-138.648, -62.365, -90.835, 44.597, 70.217, -18.455]
  MoveL 260 to (-31.45, 36.73, 22.23) mm, rotated rx -180 ry 0 rz 180 deg; joints [-138.648, -62.365, -90.835, 44.597, 70.217, -18.455]
  Call Extruder(143.84491)
  MoveL 261 to (-31.26, 36.67, 22.23) mm, rotated rx -180 ry 0 rz 180 deg; joints [-138.676, -62.369, -90.819, 44.572, 70.199, -18.455]
  MoveL 262 to (-31.26, 36.67, 22.23) mm, rotated rx -180 ry 0 rz 180 deg; joints [-138.676, -62.369, -90.819, 44.572, 70.199, -18.455]
  Call Extruder(144.07969)
  MoveL 263 to (-31.07, 36.61, 22.23) mm, rotated rx 180 ry 0 rz 180 deg; joints [-138.704, -62.373, -90.802, 44.548, 70.181, -18.455]
  MoveL 264 to (-31.07, 36.61, 22.23) mm, rotated rx 180 ry 0 rz 180 deg; joints [-138.704, -62.373, -90.802, 44.548, 70.181, -18.455]
  Call Extruder(144.31341)
  MoveL 265 to (-30.88, 36.55, 22.23) mm, rotated rx 180 ry 0 rz -180 deg; joints [-138.732, -62.377, -90.785, 44.523, 70.164, -18.455]
  MoveL 266 to (-30.88, 36.55, 22.23) mm, rotated rx 180 ry 0 rz -180 deg; joints [-138.732, -62.377, -90.785, 44.523, 70.164, -18.455]
  Call Extruder(144.54609)
  MoveL 267 to (-30.69, 36.49, 22.23) mm, rotated rx 180 ry 0 rz 180 deg; joints [-138.759, -62.381, -90.768, 44.498, 70.146, -18.455]
  MoveL 268 to (-30.69, 36.49, 22.23) mm, rotated rx 180 ry 0 rz 180 deg; joints [-138.759, -62.381, -90.768, 44.498, 70.146, -18.455]
  Call Extruder(144.81901)
  MoveL 269 to (-30.47, 36.42, 22.22) mm, rotated rx -180 ry 0 rz 180 deg; joints [-138.792, -62.386, -90.748, 44.469, 70.124, -18.456]
  MoveL 270 to (-30.47, 36.42, 22.22) mm, rotated rx -180 ry 0 rz 180 deg; joints [-138.792, -62.386, -90.748, 44.469, 70.124, -18.456]
  Call Extruder(145.09061)
  MoveL 271 to (-30.25, 36.35, 22.23) mm, rotated rx 180 ry 0 rz -180 deg; joints [-138.824, -62.391, -90.727, 44.441, 70.103, -18.456]
  MoveL 272 to (-30.25, 36.35, 22.23) mm, rotated rx 180 ry 0 rz -180 deg; joints [-138.824, -62.391, -90.727, 44.441, 70.103, -18.456]
  Call Extruder(145.36086)
  MoveL 273 to (-30.02, 36.28, 22.23) mm, rotated rx -180 ry 0 rz 180 deg; joints [-138.856, -62.396, -90.707, 44.412, 70.082, -18.457]
  MoveL 274 to (-30.02, 36.28, 22.23) mm, rotated rx -180 ry 0 rz 180 deg; joints [-138.856, -62.396, -90.707, 44.412, 70.082, -18.457]
  Call Extruder(145.62979)
  MoveL 275 to (-29.8, 36.22, 22.23) mm, rotated rx 180 ry 0 rz -180 deg; joints [-138.889, -62.401, -90.686, 44.383, 70.06, -18.457]
  MoveL 276 to (-29.8, 36.22, 22.23) mm, rotated rx 180 ry 0 rz -180 deg; joints [-138.889, -62.401, -90.686, 44.383, 70.06, -18.457]
  Call Extruder(145.88314)
  MoveL 277 to (-29.59, 36.16, 22.22) mm, rotated rx -180 ry 0 rz 180 deg; joints [-138.919, -62.406, -90.666, 44.357, 70.04, -18.459]
  MoveL 278 to (-29.59, 36.16, 22.22) mm, rotated rx -180 ry 0 rz 180 deg; joints [-138.919, -62.406, -90.666, 44.357, 70.04, -18.459]
  Call Extruder(146.12159)
  MoveL 279 to (-29.38, 36.12, 22.23) mm, rotated rx 180 ry 0 rz -180 deg; joints [-138.946, -62.411, -90.645, 44.334, 70.02, -18.461]
  MoveL 280 to (-29.38, 36.12, 22.23) mm, rotated rx 180 ry 0 rz -180 deg; joints [-138.946, -62.411, -90.645, 44.334, 70.02, -18.461]
  Call Extruder(146.35896)
  MoveL 281 to (-29.18, 36.07, 22.22) mm, rotated rx -180 ry 0 rz 180 deg; joints [-138.973, -62.416, -90.624, 44.31, 70, -18.463]
  MoveL 282 to (-29.18, 36.07, 22.22) mm, rotated rx -180 ry 0 rz 180 deg; joints [-138.973, -62.416, -90.624, 44.31, 70, -18.463]
  Call Extruder(146.59526)
  MoveL 283 to (-28.97, 36.03, 22.23) mm, rotated rx 180 ry 0 rz -180 deg; joints [-139, -62.421, -90.604, 44.286, 69.98, -18.465]
  MoveL 284 to (-28.97, 36.03, 22.23) mm, rotated rx 180 ry 0 rz -180 deg; joints [-139, -62.421, -90.604, 44.286, 69.98, -18.465]
  Call Extruder(146.83050)
  MoveL 285 to (-28.77, 35.98, 22.23) mm, rotated rx 180 ry 0 rz 180 deg; joints [-139.028, -62.426, -90.583, 44.263, 69.96, -18.468]
  MoveL 286 to (-28.77, 35.98, 22.23) mm, rotated rx 180 ry 0 rz 180 deg; joints [-139.028, -62.426, -90.583, 44.263, 69.96, -18.468]
  Call Extruder(147.11443)
  MoveL 287 to (-28.52, 35.93, 22.23) mm, rotated rx -180 ry 0 rz 180 deg; joints [-139.06, -62.432, -90.557, 44.235, 69.936, -18.471]
  MoveL 288 to (-28.52, 35.93, 22.23) mm, rotated rx -180 ry 0 rz 180 deg; joints [-139.06, -62.432, -90.557, 44.235, 69.936, -18.471]
  Call Extruder(147.39692)
  MoveL 289 to (-28.27, 35.88, 22.23) mm, rotated rx 180 ry 0 rz -180 deg; joints [-139.093, -62.438, -90.531, 44.207, 69.912, -18.474]
  MoveL 290 to (-28.27, 35.88, 22.23) mm, rotated rx 180 ry 0 rz -180 deg; joints [-139.093, -62.438, -90.531, 44.207, 69.912, -18.474]
  Call Extruder(147.67798)
  MoveL 291 to (-28.02, 35.83, 22.23) mm, rotated rx 180 ry 0 rz 180 deg; joints [-139.126, -62.445, -90.505, 44.179, 69.887, -18.477]
  MoveL 292 to (-28.02, 35.83, 22.23) mm, rotated rx 180 ry 0 rz 180 deg; joints [-139.126, -62.445, -90.505, 44.179, 69.887, -18.477]
  Call Extruder(147.95760)
  MoveL 293 to (-27.77, 35.78, 22.23) mm, rotated rx 180 ry 0 rz 180 deg; joints [-139.158, -62.451, -90.48, 44.151, 69.863, -18.481]
  MoveL 294 to (-27.77, 35.78, 22.23) mm, rotated rx 180 ry 0 rz 180 deg; joints [-139.158, -62.451, -90.48, 44.151, 69.863, -18.481]
  Call Extruder(148.23578)
  MoveL 295 to (-27.53, 35.73, 22.23) mm, rotated rx 180 ry 0 rz 180 deg; joints [-139.19, -62.457, -90.454, 44.123, 69.839, -18.484]
  MoveL 296 to (-27.53, 35.73, 22.23) mm, rotated rx 180 ry 0 rz 180 deg; joints [-139.19, -62.457, -90.454, 44.123, 69.839, -18.484]
  Call Extruder(148.51252)
  MoveL 297 to (-27.28, 35.69, 22.23) mm, rotated rx 180 ry 0 rz -180 deg; joints [-139.223, -62.464, -90.428, 44.096, 69.814, -18.487]
  MoveL 298 to (-27.28, 35.69, 22.23) mm, rotated rx 180 ry 0 rz -180 deg; joints [-139.223, -62.464, -90.428, 44.096, 69.814, -18.487]
  Call Extruder(148.72072)
  MoveL 299 to (-27.09, 35.65, 22.23) mm, rotated rx 180 ry 0 rz 180 deg; joints [-139.247, -62.468, -90.408, 44.075, 69.796, -18.489]
  MoveL 300 to (-27.09, 35.65, 22.23) mm, rotated rx 180 ry 0 rz 180 deg; joints [-139.247, -62.468, -90.408, 44.075, 69.796, -18.489]
  Call Extruder(148.95842)
  MoveL 301 to (-26.87, 35.61, 22.23) mm, rotated rx -180 ry 0 rz -180 deg; joints [-139.275, -62.474, -90.385, 44.052, 69.774, -18.493]
  MoveL 302 to (-26.87, 35.61, 22.23) mm, rotated rx -180 ry 0 rz -180 deg; joints [-139.275, -62.474, -90.385, 44.052, 69.774, -18.493]
  Call Extruder(149.29181)
  MoveL 303 to (-26.57, 35.56, 22.23) mm, rotated rx 180 ry 0 rz -180 deg; joints [-139.313, -62.482, -90.352, 44.019, 69.744, -18.498]
  MoveL 304 to (-26.57, 35.56, 22.23) mm, rotated rx 180 ry 0 rz -180 deg; joints [-139.313, -62.482, -90.352, 44.019, 69.744, -18.498]
  Call Extruder(149.62348)
  MoveL 305 to (-26.26, 35.51, 22.23) mm, rotated rx 180 ry 0 rz 180 deg; joints [-139.351, -62.49, -90.318, 43.987, 69.714, -18.503]
  MoveL 306 to (-26.26, 35.51, 22.23) mm, rotated rx 180 ry 0 rz 180 deg; joints [-139.351, -62.49, -90.318, 43.987, 69.714, -18.503]
  Call Extruder(149.95342)
  MoveL 307 to (-25.96, 35.46, 22.23) mm, rotated rx -180 ry 0 rz 180 deg; joints [-139.39, -62.498, -90.285, 43.955, 69.684, -18.509]
  MoveL 308 to (-25.96, 35.46, 22.23) mm, rotated rx -180 ry 0 rz 180 deg; joints [-139.39, -62.498, -90.285, 43.955, 69.684, -18.509]
  Call Extruder(150.28165)
  MoveL 309 to (-25.65, 35.42, 22.23) mm, rotated rx -180 ry 0 rz -180 deg; joints [-139.428, -62.507, -90.252, 43.923, 69.653, -18.514]
  MoveL 310 to (-25.65, 35.42, 22.23) mm, rotated rx -180 ry 0 rz -180 deg; joints [-139.428, -62.507, -90.252, 43.923, 69.653, -18.514]
  Call Extruder(150.60817)
  MoveL 311 to (-25.34, 35.37, 22.23) mm, rotated rx 180 ry 0 rz 180 deg; joints [-139.466, -62.515, -90.218, 43.891, 69.623, -18.519]
  MoveL 312 to (-25.34, 35.37, 22.23) mm, rotated rx 180 ry 0 rz 180 deg; joints [-139.466, -62.515, -90.218, 43.891, 69.623, -18.519]
  Call Extruder(150.97524)
  MoveL 313 to (-25, 35.32, 22.23) mm, rotated rx -180 ry 0 rz -180 deg; joints [-139.508, -62.524, -90.179, 43.856, 69.589, -18.526]
  MoveL 314 to (-25, 35.32, 22.23) mm, rotated rx -180 ry 0 rz -180 deg; joints [-139.508, -62.524, -90.179, 43.856, 69.589, -18.526]
  Call Extruder(151.38268)
  MoveL 315 to (-24.61, 35.28, 22.23) mm, rotated rx 180 ry 0 rz 180 deg; joints [-139.554, -62.535, -90.135, 43.817, 69.55, -18.534]
  MoveL 316 to (-24.61, 35.28, 22.23) mm, rotated rx 180 ry 0 rz 180 deg; joints [-139.554, -62.535, -90.135, 43.817, 69.55, -18.534]
  Call Extruder(151.78808)
  MoveL 317 to (-24.22, 35.23, 22.23) mm, rotated rx 180 ry 0 rz 180 deg; joints [-139.6, -62.546, -90.091, 43.779, 69.511, -18.542]
  MoveL 318 to (-24.22, 35.23, 22.23) mm, rotated rx 180 ry 0 rz 180 deg; joints [-139.6, -62.546, -90.091, 43.779, 69.511, -18.542]
  Call Extruder(152.19142)
  MoveL 319 to (-23.83, 35.18, 22.22) mm, rotated rx 180 ry 0 rz 180 deg; joints [-139.647, -62.557, -90.047, 43.741, 69.472, -18.551]
  MoveL 320 to (-23.83, 35.18, 22.22) mm, rotated rx 180 ry 0 rz 180 deg; joints [-139.647, -62.557, -90.047, 43.741, 69.472, -18.551]
  Call Extruder(152.59271)
  MoveL 321 to (-23.45, 35.14, 22.23) mm, rotated rx 180 ry 0 rz 180 deg; joints [-139.693, -62.568, -90.002, 43.703, 69.434, -18.559]
  MoveL 322 to (-23.45, 35.14, 22.23) mm, rotated rx 180 ry 0 rz 180 deg; joints [-139.693, -62.568, -90.002, 43.703, 69.434, -18.559]
  Call Extruder(153.19759)
  MoveL 323 to (-22.86, 35.09, 22.23) mm, rotated rx 180 ry 0 rz 180 deg; joints [-139.76, -62.586, -89.932, 43.649, 69.374, -18.574]
  MoveL 324 to (-22.86, 35.09, 22.23) mm, rotated rx 180 ry 0 rz 180 deg; joints [-139.76, -62.586, -89.932, 43.649, 69.374, -18.574]
  Call Extruder(153.79932)
  MoveL 325 to (-22.27, 35.04, 22.22) mm, rotated rx 180 ry 0 rz 180 deg; joints [-139.826, -62.603, -89.862, 43.595, 69.315, -18.589]
  MoveL 326 to (-22.27, 35.04, 22.22) mm, rotated rx 180 ry 0 rz 180 deg; joints [-139.826, -62.603, -89.862, 43.595, 69.315, -18.589]
  Call Extruder(154.39790)
  MoveL 327 to (-21.68, 35, 22.22) mm, rotated rx -180 ry 0 rz -180 deg; joints [-139.893, -62.62, -89.792, 43.541, 69.255, -18.604]
  MoveL 328 to (-21.68, 35, 22.22) mm, rotated rx -180 ry 0 rz -180 deg; joints [-139.893, -62.62, -89.792, 43.541, 69.255, -18.604]
  Call Extruder(155.56967)
  MoveL 329 to (-20.52, 34.95, 22.22) mm, rotated rx -180 ry 0 rz -180 deg; joints [-140.019, -62.657, -89.648, 43.442, 69.137, -18.638]
  MoveL 330 to (-20.52, 34.95, 22.22) mm, rotated rx -180 ry 0 rz -180 deg; joints [-140.019, -62.657, -89.648, 43.442, 69.137, -18.638]
  Call Extruder(157.02754)
  MoveL 331 to (-19.06, 34.91, 22.23) mm, rotated rx 180 ry 0 rz 180 deg; joints [-140.173, -62.703, -89.465, 43.322, 68.988, -18.683]
  Call Extruder(395.62063)
  MoveL 332 to (219.06, 34.91, 22.23) mm, rotated rx 180 ry 0 rz -180 deg; joints [-155.896, -78.433, -46.554, 37.963, 41.596, -30.264]
  Call Extruder(396.49572)
  MoveL 333 to (219.94, 34.93, 22.23) mm, rotated rx 180 ry 0 rz 180 deg; joints [-155.931, -78.533, -46.328, 38.007, 41.478, -30.348]
  MoveL 334 to (219.94, 34.93, 22.23) mm, rotated rx 180 ry 0 rz 180 deg; joints [-155.931, -78.533, -46.328, 38.007, 41.478, -30.348]
  Call Extruder(397.66749)
  MoveL 335 to (221.1, 34.97, 22.23) mm, rotated rx 180 ry 0 rz 180 deg; joints [-155.975, -78.667, -46.022, 38.069, 41.322, -30.465]
  MoveL 336 to (221.1, 34.97, 22.23) mm, rotated rx 180 ry 0 rz 180 deg; joints [-155.975, -78.667, -46.022, 38.069, 41.322, -30.465]
  Call Extruder(398.55557)
  MoveL 337 to (221.97, 35.02, 22.22) mm, rotated rx 180 ry 0 rz -180 deg; joints [-156.007, -78.77, -45.789, 38.119, 41.203, -30.555]
  MoveL 338 to (221.97, 35.02, 22.22) mm, rotated rx 180 ry 0 rz -180 deg; joints [-156.007, -78.77, -45.789, 38.119, 41.203, -30.555]
  Call Extruder(399.15730)
  MoveL 339 to (222.56, 35.07, 22.23) mm, rotated rx 180 ry 0 rz -180 deg; joints [-156.027, -78.84, -45.63, 38.155, 41.123, -30.619]
  MoveL 340 to (222.56, 35.07, 22.23) mm, rotated rx 180 ry 0 rz -180 deg; joints [-156.027, -78.84, -45.63, 38.155, 41.123, -30.619]
  Call Extruder(399.76217)
  MoveL 341 to (223.15, 35.11, 22.23) mm, rotated rx -180 ry 0 rz 180 deg; joints [-156.047, -78.911, -45.471, 38.192, 41.043, -30.683]
  MoveL 342 to (223.15, 35.11, 22.23) mm, rotated rx -180 ry 0 rz 180 deg; joints [-156.047, -78.911, -45.471, 38.192, 41.043, -30.683]
  Call Extruder(400.26672)
  MoveL 343 to (223.64, 35.16, 22.23) mm, rotated rx 180 ry 0 rz 180 deg; joints [-156.062, -78.969, -45.338, 38.225, 40.976, -30.737]
  MoveL 344 to (223.64, 35.16, 22.23) mm, rotated rx 180 ry 0 rz 180 deg; joints [-156.062, -78.969, -45.338, 38.225, 40.976, -30.737]
  Call Extruder(400.67007)
  MoveL 345 to (224.03, 35.21, 22.23) mm, rotated rx -180 ry 0 rz 180 deg; joints [-156.074, -79.017, -45.231, 38.252, 40.923, -30.782]
  MoveL 346 to (224.03, 35.21, 22.23) mm, rotated rx -180 ry 0 rz 180 deg; joints [-156.074, -79.017, -45.231, 38.252, 40.923, -30.782]
  Call Extruder(401.07546)
  MoveL 347 to (224.42, 35.25, 22.23) mm, rotated rx -180 ry 0 rz 180 deg; joints [-156.086, -79.064, -45.123, 38.279, 40.871, -30.827]
  MoveL 348 to (224.42, 35.25, 22.23) mm, rotated rx -180 ry 0 rz 180 deg; joints [-156.086, -79.064, -45.123, 38.279, 40.871, -30.827]
  Call Extruder(401.48291)
  MoveL 349 to (224.8, 35.3, 22.22) mm, rotated rx -180 ry 0 rz 180 deg; joints [-156.097, -79.112, -45.016, 38.307, 40.818, -30.872]
  MoveL 350 to (224.8, 35.3, 22.22) mm, rotated rx -180 ry 0 rz 180 deg; joints [-156.097, -79.112, -45.016, 38.307, 40.818, -30.872]
  Call Extruder(401.89240)
  MoveL 351 to (225.19, 35.34, 22.22) mm, rotated rx 180 ry 0 rz 180 deg; joints [-156.109, -79.159, -44.908, 38.335, 40.765, -30.918]
  MoveL 352 to (225.19, 35.34, 22.22) mm, rotated rx 180 ry 0 rz 180 deg; joints [-156.109, -79.159, -44.908, 38.335, 40.765, -30.918]
  Call Extruder(402.21894)
  MoveL 353 to (225.5, 35.39, 22.23) mm, rotated rx -180 ry 0 rz 180 deg; joints [-156.117, -79.198, -44.822, 38.359, 40.723, -30.956]
  MoveL 354 to (225.5, 35.39, 22.23) mm, rotated rx -180 ry 0 rz 180 deg; joints [-156.117, -79.198, -44.822, 38.359, 40.723, -30.956]
  Call Extruder(402.54719)
  MoveL 355 to (225.8, 35.44, 22.23) mm, rotated rx -180 ry 0 rz 180 deg; joints [-156.125, -79.236, -44.735, 38.384, 40.681, -30.994]
  MoveL 356 to (225.8, 35.44, 22.23) mm, rotated rx -180 ry 0 rz 180 deg; joints [-156.125, -79.236, -44.735, 38.384, 40.681, -30.994]
  Call Extruder(402.87716)
  MoveL 357 to (226.11, 35.49, 22.22) mm, rotated rx -180 ry 0 rz 180 deg; joints [-156.133, -79.275, -44.649, 38.408, 40.639, -31.032]
  MoveL 358 to (226.11, 35.49, 22.22) mm, rotated rx -180 ry 0 rz 180 deg; joints [-156.133, -79.275, -44.649, 38.408, 40.639, -31.032]
  Call Extruder(403.20885)
  MoveL 359 to (226.41, 35.54, 22.23) mm, rotated rx 180 ry 0 rz -180 deg; joints [-156.141, -79.313, -44.562, 38.432, 40.597, -31.07]
  MoveL 360 to (226.41, 35.54, 22.23) mm, rotated rx 180 ry 0 rz -180 deg; joints [-156.141, -79.313, -44.562, 38.432, 40.597, -31.07]
  Call Extruder(403.54226)
  MoveL 361 to (226.72, 35.59, 22.23) mm, rotated rx 180 ry 0 rz -180 deg; joints [-156.149, -79.352, -44.474, 38.457, 40.555, -31.108]
  MoveL 362 to (226.72, 35.59, 22.23) mm, rotated rx 180 ry 0 rz -180 deg; joints [-156.149, -79.352, -44.474, 38.457, 40.555, -31.108]
  Call Extruder(403.87738)
  MoveL 363 to (227.03, 35.63, 22.23) mm, rotated rx -180 ry 0 rz 180 deg; joints [-156.157, -79.39, -44.387, 38.482, 40.513, -31.146]
  MoveL 364 to (227.03, 35.63, 22.23) mm, rotated rx -180 ry 0 rz 180 deg; joints [-156.157, -79.39, -44.387, 38.482, 40.513, -31.146]
  Call Extruder(404.15384)
  MoveL 365 to (227.27, 35.68, 22.22) mm, rotated rx -180 ry 0 rz -180 deg; joints [-156.162, -79.423, -44.315, 38.504, 40.478, -31.179]
  MoveL 366 to (227.27, 35.68, 22.22) mm, rotated rx -180 ry 0 rz -180 deg; joints [-156.162, -79.423, -44.315, 38.504, 40.478, -31.179]
  Call Extruder(404.43174)
  MoveL 367 to (227.52, 35.73, 22.23) mm, rotated rx 180 ry 0 rz -180 deg; joints [-156.168, -79.455, -44.243, 38.526, 40.444, -31.212]
  MoveL 368 to (227.52, 35.73, 22.23) mm, rotated rx 180 ry 0 rz -180 deg; joints [-156.168, -79.455, -44.243, 38.526, 40.444, -31.212]
  Call Extruder(404.71108)
  MoveL 369 to (227.77, 35.78, 22.23) mm, rotated rx -180 ry 0 rz -180 deg; joints [-156.173, -79.487, -44.17, 38.548, 40.41, -31.246]
  MoveL 370 to (227.77, 35.78, 22.23) mm, rotated rx -180 ry 0 rz -180 deg; joints [-156.173, -79.487, -44.17, 38.548, 40.41, -31.246]
  Call Extruder(404.99186)
  MoveL 371 to (228.02, 35.83, 22.23) mm, rotated rx 180 ry 0 rz 180 deg; joints [-156.179, -79.519, -44.098, 38.57, 40.375, -31.279]
  MoveL 372 to (228.02, 35.83, 22.23) mm, rotated rx 180 ry 0 rz 180 deg; joints [-156.179, -79.519, -44.098, 38.57, 40.375, -31.279]
  Call Extruder(405.27408)
  MoveL 373 to (228.27, 35.88, 22.23) mm, rotated rx 180 ry 0 rz -180 deg; joints [-156.185, -79.551, -44.025, 38.592, 40.341, -31.312]
  MoveL 374 to (228.27, 35.88, 22.23) mm, rotated rx 180 ry 0 rz -180 deg; joints [-156.185, -79.551, -44.025, 38.592, 40.341, -31.312]
  Call Extruder(405.55775)
  MoveL 375 to (228.52, 35.93, 22.22) mm, rotated rx 180 ry 0 rz -180 deg; joints [-156.19, -79.584, -43.952, 38.615, 40.307, -31.345]
  MoveL 376 to (228.52, 35.93, 22.22) mm, rotated rx 180 ry 0 rz -180 deg; joints [-156.19, -79.584, -43.952, 38.615, 40.307, -31.345]
  Call Extruder(405.84286)
  MoveL 377 to (228.77, 35.98, 22.23) mm, rotated rx -180 ry 0 rz -180 deg; joints [-156.196, -79.616, -43.88, 38.637, 40.272, -31.379]
  MoveL 378 to (228.77, 35.98, 22.23) mm, rotated rx -180 ry 0 rz -180 deg; joints [-156.196, -79.616, -43.88, 38.637, 40.272, -31.379]
  Call Extruder(406.07863)
  MoveL 379 to (228.97, 36.03, 22.22) mm, rotated rx 180 ry 0 rz 180 deg; joints [-156.2, -79.643, -43.819, 38.656, 40.244, -31.407]
  MoveL 380 to (228.97, 36.03, 22.22) mm, rotated rx 180 ry 0 rz 180 deg; joints [-156.2, -79.643, -43.819, 38.656, 40.244, -31.407]
  Call Extruder(406.31548)
  MoveL 381 to (229.18, 36.07, 22.23) mm, rotated rx 180 ry 0 rz 180 deg; joints [-156.204, -79.67, -43.759, 38.676, 40.215, -31.435]
  MoveL 382 to (229.18, 36.07, 22.23) mm, rotated rx 180 ry 0 rz 180 deg; joints [-156.204, -79.67, -43.759, 38.676, 40.215, -31.435]
  Call Extruder(406.55339)
  MoveL 383 to (229.38, 36.12, 22.23) mm, rotated rx 180 ry 0 rz -180 deg; joints [-156.208, -79.697, -43.699, 38.695, 40.187, -31.463]
  MoveL 384 to (229.38, 36.12, 22.23) mm, rotated rx 180 ry 0 rz -180 deg; joints [-156.208, -79.697, -43.699, 38.695, 40.187, -31.463]
  Call Extruder(406.79238)
  MoveL 385 to (229.59, 36.16, 22.22) mm, rotated rx -180 ry 0 rz -180 deg; joints [-156.212, -79.724, -43.638, 38.714, 40.159, -31.491]
  MoveL 386 to (229.59, 36.16, 22.22) mm, rotated rx -180 ry 0 rz -180 deg; joints [-156.212, -79.724, -43.638, 38.714, 40.159, -31.491]
  Call Extruder(407.04637)
  MoveL 387 to (229.8, 36.22, 22.22) mm, rotated rx -180 ry 0 rz 180 deg; joints [-156.216, -79.752, -43.574, 38.736, 40.129, -31.523]
  MoveL 388 to (229.8, 36.22, 22.22) mm, rotated rx -180 ry 0 rz 180 deg; joints [-156.216, -79.752, -43.574, 38.736, 40.129, -31.523]
  Call Extruder(407.31597)
  MoveL 389 to (230.02, 36.28, 22.22) mm, rotated rx -180 ry 0 rz -180 deg; joints [-156.219, -79.783, -43.505, 38.761, 40.098, -31.557]
  MoveL 390 to (230.02, 36.28, 22.22) mm, rotated rx -180 ry 0 rz -180 deg; joints [-156.219, -79.783, -43.505, 38.761, 40.098, -31.557]
  Call Extruder(407.58690)
  MoveL 391 to (230.25, 36.35, 22.22) mm, rotated rx 180 ry 0 rz 180 deg; joints [-156.221, -79.814, -43.437, 38.785, 40.067, -31.591]
  MoveL 392 to (230.25, 36.35, 22.22) mm, rotated rx 180 ry 0 rz 180 deg; joints [-156.221, -79.814, -43.437, 38.785, 40.067, -31.591]
  Call Extruder(407.85917)
  MoveL 393 to (230.47, 36.42, 22.23) mm, rotated rx 180 ry 0 rz 180 deg; joints [-156.224, -79.844, -43.368, 38.81, 40.036, -31.625]
  MoveL 394 to (230.47, 36.42, 22.23) mm, rotated rx 180 ry 0 rz 180 deg; joints [-156.224, -79.844, -43.368, 38.81, 40.036, -31.625]
  Call Extruder(408.13278)
  MoveL 395 to (230.69, 36.49, 22.23) mm, rotated rx 180 ry 0 rz -180 deg; joints [-156.227, -79.875, -43.299, 38.834, 40.005, -31.659]
  MoveL 396 to (230.69, 36.49, 22.23) mm, rotated rx 180 ry 0 rz -180 deg; joints [-156.227, -79.875, -43.299, 38.834, 40.005, -31.659]
  Call Extruder(408.36597)
  MoveL 397 to (230.88, 36.55, 22.23) mm, rotated rx -180 ry 0 rz 180 deg; joints [-156.229, -79.901, -43.24, 38.856, 39.978, -31.689]
  MoveL 398 to (230.88, 36.55, 22.23) mm, rotated rx -180 ry 0 rz 180 deg; joints [-156.229, -79.901, -43.24, 38.856, 39.978, -31.689]
  Call Extruder(408.60021)
  MoveL 399 to (231.07, 36.61, 22.22) mm, rotated rx -180 ry 0 rz 180 deg; joints [-156.231, -79.927, -43.182, 38.878, 39.952, -31.719]
  MoveL 400 to (231.07, 36.61, 22.22) mm, rotated rx -180 ry 0 rz 180 deg; joints [-156.231, -79.927, -43.182, 38.878, 39.952, -31.719]
  Call Extruder(408.83551)
  MoveL 401 to (231.26, 36.67, 22.23) mm, rotated rx 180 ry 0 rz 180 deg; joints [-156.233, -79.954, -43.123, 38.899, 39.926, -31.748]
  MoveL 402 to (231.26, 36.67, 22.23) mm, rotated rx 180 ry 0 rz 180 deg; joints [-156.233, -79.954, -43.123, 38.899, 39.926, -31.748]
  Call Extruder(409.07185)
  MoveL 403 to (231.45, 36.73, 22.23) mm, rotated rx 180 ry 0 rz 180 deg; joints [-156.235, -79.98, -43.064, 38.921, 39.899, -31.778]
  MoveL 404 to (231.45, 36.73, 22.23) mm, rotated rx 180 ry 0 rz 180 deg; joints [-156.235, -79.98, -43.064, 38.921, 39.899, -31.778]
  Call Extruder(409.30925)
  MoveL 405 to (231.64, 36.79, 22.22) mm, rotated rx 180 ry 0 rz 180 deg; joints [-156.237, -80.006, -43.006, 38.943, 39.873, -31.808]
  MoveL 406 to (231.64, 36.79, 22.22) mm, rotated rx 180 ry 0 rz 180 deg; joints [-156.237, -80.006, -43.006, 38.943, 39.873, -31.808]
  Call Extruder(409.68944)
  MoveL 407 to (231.93, 36.91, 22.23) mm, rotated rx 180 ry 0 rz 180 deg; joints [-156.238, -80.048, -42.911, 38.981, 39.832, -31.858]
  MoveL 408 to (231.93, 36.91, 22.23) mm, rotated rx 180 ry 0 rz 180 deg; joints [-156.238, -80.048, -42.911, 38.981, 39.832, -31.858]
  Call Extruder(410.07143)
  MoveL 409 to (232.22, 37.03, 22.22) mm, rotated rx 180 ry 0 rz 180 deg; joints [-156.238, -80.091, -42.817, 39.02, 39.791, -31.909]
  MoveL 410 to (232.22, 37.03, 22.22) mm, rotated rx 180 ry 0 rz 180 deg; joints [-156.238, -80.091, -42.817, 39.02, 39.791, -31.909]
  Call Extruder(410.42789)
  MoveL 411 to (232.49, 37.15, 22.23) mm, rotated rx -180 ry 0 rz 180 deg; joints [-156.239, -80.13, -42.729, 39.056, 39.753, -31.956]
  MoveL 412 to (232.49, 37.15, 22.23) mm, rotated rx -180 ry 0 rz 180 deg; joints [-156.239, -80.13, -42.729, 39.056, 39.753, -31.956]
  Call Extruder(410.75854)
  MoveL 413 to (232.74, 37.26, 22.22) mm, rotated rx 180 ry 0 rz 180 deg; joints [-156.239, -80.166, -42.648, 39.09, 39.718, -32]
  MoveL 414 to (232.74, 37.26, 22.22) mm, rotated rx 180 ry 0 rz 180 deg; joints [-156.239, -80.166, -42.648, 39.09, 39.718, -32]
  Call Extruder(411.09062)
  MoveL 415 to (232.99, 37.36, 22.22) mm, rotated rx 180 ry 0 rz -180 deg; joints [-156.239, -80.203, -42.566, 39.124, 39.683, -32.045]
  MoveL 416 to (232.99, 37.36, 22.22) mm, rotated rx 180 ry 0 rz -180 deg; joints [-156.239, -80.203, -42.566, 39.124, 39.683, -32.045]
  Call Extruder(411.52249)
  MoveL 417 to (233.29, 37.54, 22.22) mm, rotated rx 180 ry 0 rz 180 deg; joints [-156.236, -80.25, -42.461, 39.173, 39.64, -32.106]
  MoveL 418 to (233.29, 37.54, 22.22) mm, rotated rx 180 ry 0 rz 180 deg; joints [-156.236, -80.25, -42.461, 39.173, 39.64, -32.106]
  Call Extruder(411.95620)
  MoveL 419 to (233.6, 37.71, 22.23) mm, rotated rx 180 ry 0 rz 180 deg; joints [-156.232, -80.297, -42.356, 39.222, 39.597, -32.167]
  MoveL 420 to (233.6, 37.71, 22.23) mm, rotated rx 180 ry 0 rz 180 deg; joints [-156.232, -80.297, -42.356, 39.222, 39.597, -32.167]
  Call Extruder(412.39175)
  MoveL 421 to (233.9, 37.89, 22.23) mm, rotated rx 180 ry 0 rz 180 deg; joints [-156.228, -80.344, -42.251, 39.271, 39.554, -32.229]
  MoveL 422 to (233.9, 37.89, 22.23) mm, rotated rx 180 ry 0 rz 180 deg; joints [-156.228, -80.344, -42.251, 39.271, 39.554, -32.229]
  Call Extruder(412.82915)
  MoveL 423 to (234.21, 38.06, 22.22) mm, rotated rx 180 ry 0 rz 180 deg; joints [-156.224, -80.392, -42.145, 39.321, 39.511, -32.291]
  MoveL 424 to (234.21, 38.06, 22.22) mm, rotated rx 180 ry 0 rz 180 deg; joints [-156.224, -80.392, -42.145, 39.321, 39.511, -32.291]
  Call Extruder(413.20589)
  MoveL 425 to (234.45, 38.24, 22.22) mm, rotated rx 180 ry 0 rz 180 deg; joints [-156.218, -80.432, -42.055, 39.367, 39.476, -32.346]
  MoveL 426 to (234.45, 38.24, 22.22) mm, rotated rx 180 ry 0 rz 180 deg; joints [-156.218, -80.432, -42.055, 39.367, 39.476, -32.346]
  Call Extruder(413.90582)
  MoveL 427 to (234.9, 38.57, 22.22) mm, rotated rx -180 ry 0 rz 180 deg; joints [-156.206, -80.506, -41.89, 39.453, 39.412, -32.449]
  MoveL 428 to (234.9, 38.57, 22.22) mm, rotated rx -180 ry 0 rz 180 deg; joints [-156.206, -80.506, -41.89, 39.453, 39.412, -32.449]
  Call Extruder(414.60855)
  MoveL 429 to (235.35, 38.9, 22.23) mm, rotated rx 180 ry 0 rz 180 deg; joints [-156.195, -80.581, -41.724, 39.54, 39.348, -32.553]
  Call Extruder(416.34741)
  MoveL 430 to (236.39, 39.81, 22.23) mm, rotated rx 180 ry 0 rz 180 deg; joints [-156.154, -80.762, -41.321, 39.767, 39.199, -32.819]
  Call Extruder(418.08626)
  MoveL 431 to (237.3, 40.85, 22.22) mm, rotated rx -180 ry 0 rz 180 deg; joints [-156.097, -80.937, -40.934, 40.01, 39.068, -33.093]
  Call Extruder(418.43762)
  MoveL 432 to (237.47, 41.07, 22.23) mm, rotated rx 180 ry 0 rz 180 deg; joints [-156.083, -80.97, -40.859, 40.061, 39.044, -33.149]
  MoveL 433 to (237.47, 41.07, 22.23) mm, rotated rx 180 ry 0 rz 180 deg; joints [-156.083, -80.97, -40.859, 40.061, 39.044, -33.149]
  Call Extruder(419.13755)
  MoveL 434 to (237.8, 41.52, 22.23) mm, rotated rx 180 ry 0 rz 180 deg; joints [-156.055, -81.038, -40.71, 40.163, 38.996, -33.262]
  MoveL 435 to (237.8, 41.52, 22.23) mm, rotated rx 180 ry 0 rz 180 deg; joints [-156.055, -81.038, -40.71, 40.163, 38.996, -33.262]
  Call Extruder(419.83467)
  MoveL 436 to (238.12, 41.98, 22.23) mm, rotated rx -180 ry 0 rz -180 deg; joints [-156.028, -81.106, -40.559, 40.265, 38.948, -33.375]
  MoveL 437 to (238.12, 41.98, 22.23) mm, rotated rx -180 ry 0 rz -180 deg; joints [-156.028, -81.106, -40.559, 40.265, 38.948, -33.375]
  Call Extruder(420.08158)
  MoveL 438 to (238.22, 42.15, 22.22) mm, rotated rx 180 ry 0 rz -180 deg; joints [-156.016, -81.128, -40.509, 40.302, 38.933, -33.415]
  MoveL 439 to (238.22, 42.15, 22.22) mm, rotated rx 180 ry 0 rz -180 deg; joints [-156.016, -81.128, -40.509, 40.302, 38.933, -33.415]
  Call Extruder(420.51713)
  MoveL 440 to (238.4, 42.45, 22.23) mm, rotated rx 180 ry 0 rz -180 deg; joints [-155.996, -81.169, -40.42, 40.368, 38.908, -33.486]
  MoveL 441 to (238.4, 42.45, 22.23) mm, rotated rx 180 ry 0 rz -180 deg; joints [-155.996, -81.169, -40.42, 40.368, 38.908, -33.486]
  Call Extruder(420.95084)
  MoveL 442 to (238.57, 42.75, 22.22) mm, rotated rx 180 ry 0 rz 180 deg; joints [-155.976, -81.209, -40.332, 40.434, 38.882, -33.557]
  MoveL 443 to (238.57, 42.75, 22.22) mm, rotated rx 180 ry 0 rz 180 deg; joints [-155.976, -81.209, -40.332, 40.434, 38.882, -33.557]
  Call Extruder(421.38271)
  MoveL 444 to (238.75, 43.06, 22.23) mm, rotated rx -180 ry 0 rz -180 deg; joints [-155.956, -81.249, -40.243, 40.5, 38.856, -33.628]
  MoveL 445 to (238.75, 43.06, 22.23) mm, rotated rx -180 ry 0 rz -180 deg; joints [-155.956, -81.249, -40.243, 40.5, 38.856, -33.628]
  Call Extruder(421.76312)
  MoveL 446 to (238.89, 43.34, 22.23) mm, rotated rx 180 ry 0 rz 180 deg; joints [-155.937, -81.283, -40.167, 40.559, 38.835, -33.691]
  MoveL 447 to (238.89, 43.34, 22.23) mm, rotated rx 180 ry 0 rz 180 deg; joints [-155.937, -81.283, -40.167, 40.559, 38.835, -33.691]
  Call Extruder(422.09380)
  MoveL 448 to (239, 43.58, 22.22) mm, rotated rx -180 ry 0 rz -180 deg; joints [-155.919, -81.312, -40.105, 40.611, 38.819, -33.745]
  MoveL 449 to (239, 43.58, 22.22) mm, rotated rx -180 ry 0 rz -180 deg; joints [-155.919, -81.312, -40.105, 40.611, 38.819, -33.745]
  Call Extruder(422.42305)
  MoveL 450 to (239.1, 43.83, 22.23) mm, rotated rx 180 ry 0 rz -180 deg; joints [-155.901, -81.34, -40.042, 40.662, 38.803, -33.799]
  MoveL 451 to (239.1, 43.83, 22.23) mm, rotated rx 180 ry 0 rz -180 deg; joints [-155.901, -81.34, -40.042, 40.662, 38.803, -33.799]
  Call Extruder(422.80503)
  MoveL 452 to (239.23, 44.12, 22.23) mm, rotated rx 180 ry 0 rz 180 deg; joints [-155.879, -81.373, -39.97, 40.722, 38.785, -33.862]
  MoveL 453 to (239.23, 44.12, 22.23) mm, rotated rx 180 ry 0 rz 180 deg; joints [-155.879, -81.373, -39.97, 40.722, 38.785, -33.862]
  Call Extruder(423.18522)
  MoveL 454 to (239.35, 44.42, 22.23) mm, rotated rx 180 ry 0 rz -180 deg; joints [-155.858, -81.405, -39.898, 40.783, 38.767, -33.925]
  MoveL 455 to (239.35, 44.42, 22.23) mm, rotated rx 180 ry 0 rz -180 deg; joints [-155.858, -81.405, -39.898, 40.783, 38.767, -33.925]
  Call Extruder(423.49290)
  MoveL 456 to (239.44, 44.66, 22.23) mm, rotated rx 180 ry 0 rz -180 deg; joints [-155.84, -81.431, -39.84, 40.832, 38.753, -33.976]
  MoveL 457 to (239.44, 44.66, 22.23) mm, rotated rx 180 ry 0 rz -180 deg; joints [-155.84, -81.431, -39.84, 40.832, 38.753, -33.976]
  Call Extruder(423.72925)
  MoveL 458 to (239.5, 44.85, 22.23) mm, rotated rx 180 ry 0 rz 180 deg; joints [-155.826, -81.45, -39.798, 40.87, 38.744, -34.015]
  MoveL 459 to (239.5, 44.85, 22.23) mm, rotated rx 180 ry 0 rz 180 deg; joints [-155.826, -81.45, -39.798, 40.87, 38.744, -34.015]
  Call Extruder(423.96455)
  MoveL 460 to (239.56, 45.03, 22.23) mm, rotated rx 180 ry 0 rz 180 deg; joints [-155.811, -81.469, -39.756, 40.907, 38.735, -34.054]
  MoveL 461 to (239.56, 45.03, 22.23) mm, rotated rx 180 ry 0 rz 180 deg; joints [-155.811, -81.469, -39.756, 40.907, 38.735, -34.054]
  Call Extruder(424.19880)
  MoveL 462 to (239.62, 45.22, 22.22) mm, rotated rx -180 ry 0 rz -180 deg; joints [-155.797, -81.489, -39.714, 40.945, 38.725, -34.093]
  MoveL 463 to (239.62, 45.22, 22.22) mm, rotated rx -180 ry 0 rz -180 deg; joints [-155.797, -81.489, -39.714, 40.945, 38.725, -34.093]
  Call Extruder(424.43200)
  MoveL 464 to (239.68, 45.41, 22.23) mm, rotated rx 180 ry 0 rz 180 deg; joints [-155.783, -81.508, -39.672, 40.983, 38.716, -34.132]
  MoveL 465 to (239.68, 45.41, 22.23) mm, rotated rx 180 ry 0 rz 180 deg; joints [-155.783, -81.508, -39.672, 40.983, 38.716, -34.132]
  Call Extruder(424.68486)
  MoveL 466 to (239.75, 45.62, 22.23) mm, rotated rx 180 ry 0 rz 180 deg; joints [-155.767, -81.528, -39.627, 41.024, 38.706, -34.174]
  MoveL 467 to (239.75, 45.62, 22.23) mm, rotated rx 180 ry 0 rz 180 deg; joints [-155.767, -81.528, -39.627, 41.024, 38.706, -34.174]
  Call Extruder(424.95712)
  MoveL 468 to (239.81, 45.84, 22.23) mm, rotated rx 180 ry 0 rz 180 deg; joints [-155.75, -81.55, -39.578, 41.069, 38.696, -34.22]
  MoveL 469 to (239.81, 45.84, 22.23) mm, rotated rx 180 ry 0 rz 180 deg; joints [-155.75, -81.55, -39.578, 41.069, 38.696, -34.22]
  Call Extruder(425.22805)
  MoveL 470 to (239.88, 46.06, 22.23) mm, rotated rx 180 ry 0 rz 180 deg; joints [-155.733, -81.572, -39.529, 41.113, 38.685, -34.265]
  MoveL 471 to (239.88, 46.06, 22.23) mm, rotated rx 180 ry 0 rz 180 deg; joints [-155.733, -81.572, -39.529, 41.113, 38.685, -34.265]
  Call Extruder(425.49763)
  MoveL 472 to (239.95, 46.29, 22.23) mm, rotated rx -180 ry 0 rz 180 deg; joints [-155.715, -81.595, -39.481, 41.158, 38.675, -34.311]
  MoveL 473 to (239.95, 46.29, 22.23) mm, rotated rx -180 ry 0 rz 180 deg; joints [-155.715, -81.595, -39.481, 41.158, 38.675, -34.311]
  Call Extruder(425.76589)
  MoveL 474 to (240.02, 46.51, 22.23) mm, rotated rx 180 ry 0 rz 180 deg; joints [-155.698, -81.617, -39.432, 41.203, 38.665, -34.357]
  MoveL 475 to (240.02, 46.51, 22.23) mm, rotated rx 180 ry 0 rz 180 deg; joints [-155.698, -81.617, -39.432, 41.203, 38.665, -34.357]
  Call Extruder(426.00483)
  MoveL 476 to (240.06, 46.72, 22.23) mm, rotated rx 180 ry 0 rz -180 deg; joints [-155.682, -81.635, -39.392, 41.242, 38.658, -34.397]
  MoveL 477 to (240.06, 46.72, 22.23) mm, rotated rx 180 ry 0 rz -180 deg; joints [-155.682, -81.635, -39.392, 41.242, 38.658, -34.397]
  Call Extruder(426.24270)
  MoveL 478 to (240.11, 46.92, 22.22) mm, rotated rx 180 ry 0 rz -180 deg; joints [-155.665, -81.653, -39.352, 41.282, 38.651, -34.437]
  MoveL 479 to (240.11, 46.92, 22.22) mm, rotated rx 180 ry 0 rz -180 deg; joints [-155.665, -81.653, -39.352, 41.282, 38.651, -34.437]
  Call Extruder(426.47950)
  MoveL 480 to (240.15, 47.12, 22.23) mm, rotated rx 180 ry 0 rz 180 deg; joints [-155.649, -81.671, -39.313, 41.321, 38.644, -34.476]
  MoveL 481 to (240.15, 47.12, 22.23) mm, rotated rx 180 ry 0 rz 180 deg; joints [-155.649, -81.671, -39.313, 41.321, 38.644, -34.476]
  Call Extruder(426.71523)
  MoveL 482 to (240.2, 47.33, 22.23) mm, rotated rx 180 ry 0 rz 180 deg; joints [-155.633, -81.689, -39.273, 41.361, 38.637, -34.516]
  MoveL 483 to (240.2, 47.33, 22.23) mm, rotated rx 180 ry 0 rz 180 deg; joints [-155.633, -81.689, -39.273, 41.361, 38.637, -34.516]
  Call Extruder(426.97511)
  MoveL 484 to (240.24, 47.55, 22.23) mm, rotated rx 180 ry 0 rz 180 deg; joints [-155.614, -81.709, -39.229, 41.404, 38.629, -34.56]
  MoveL 485 to (240.24, 47.55, 22.23) mm, rotated rx 180 ry 0 rz 180 deg; joints [-155.614, -81.709, -39.229, 41.404, 38.629, -34.56]
  Call Extruder(427.25877)
  MoveL 486 to (240.29, 47.8, 22.23) mm, rotated rx 180 ry 0 rz 180 deg; joints [-155.594, -81.73, -39.182, 41.452, 38.621, -34.608]
  MoveL 487 to (240.29, 47.8, 22.23) mm, rotated rx 180 ry 0 rz 180 deg; joints [-155.594, -81.73, -39.182, 41.452, 38.621, -34.608]
  Call Extruder(427.54099)
  MoveL 488 to (240.34, 48.05, 22.23) mm, rotated rx 180 ry 0 rz -180 deg; joints [-155.574, -81.752, -39.135, 41.5, 38.613, -34.656]
  MoveL 489 to (240.34, 48.05, 22.23) mm, rotated rx 180 ry 0 rz -180 deg; joints [-155.574, -81.752, -39.135, 41.5, 38.613, -34.656]
  Call Extruder(427.82177)
  MoveL 490 to (240.39, 48.3, 22.22) mm, rotated rx -180 ry 0 rz 180 deg; joints [-155.554, -81.773, -39.087, 41.548, 38.605, -34.705]
  MoveL 491 to (240.39, 48.3, 22.22) mm, rotated rx -180 ry 0 rz 180 deg; joints [-155.554, -81.773, -39.087, 41.548, 38.605, -34.705]
  Call Extruder(428.10111)
  MoveL 492 to (240.44, 48.55, 22.22) mm, rotated rx -180 ry 0 rz 180 deg; joints [-155.534, -81.795, -39.04, 41.596, 38.598, -34.753]
  MoveL 493 to (240.44, 48.55, 22.22) mm, rotated rx -180 ry 0 rz 180 deg; joints [-155.534, -81.795, -39.04, 41.596, 38.598, -34.753]
  Call Extruder(428.37901)
  MoveL 494 to (240.49, 48.8, 22.23) mm, rotated rx -180 ry 0 rz 180 deg; joints [-155.514, -81.817, -38.992, 41.644, 38.59, -34.801]
  MoveL 495 to (240.49, 48.8, 22.23) mm, rotated rx -180 ry 0 rz 180 deg; joints [-155.514, -81.817, -38.992, 41.644, 38.59, -34.801]
  Call Extruder(428.65546)
  MoveL 496 to (240.54, 49.05, 22.23) mm, rotated rx 180 ry 0 rz 180 deg; joints [-155.494, -81.838, -38.945, 41.692, 38.582, -34.849]
  MoveL 497 to (240.54, 49.05, 22.23) mm, rotated rx 180 ry 0 rz 180 deg; joints [-155.494, -81.838, -38.945, 41.692, 38.582, -34.849]
  Call Extruder(428.96049)
  MoveL 498 to (240.59, 49.33, 22.23) mm, rotated rx 180 ry 0 rz 180 deg; joints [-155.471, -81.861, -38.894, 41.745, 38.574, -34.902]
  MoveL 499 to (240.59, 49.33, 22.23) mm, rotated rx 180 ry 0 rz 180 deg; joints [-155.471, -81.861, -38.894, 41.745, 38.574, -34.902]
  Call Extruder(429.29393)
  MoveL 500 to (240.64, 49.63, 22.23) mm, rotated rx 180 ry 0 rz -180 deg; joints [-155.446, -81.887, -38.839, 41.803, 38.566, -34.96]
  MoveL 501 to (240.64, 49.63, 22.23) mm, rotated rx 180 ry 0 rz -180 deg; joints [-155.446, -81.887, -38.839, 41.803, 38.566, -34.96]
  Call Extruder(429.62565)
  MoveL 502 to (240.69, 49.94, 22.22) mm, rotated rx -180 ry 0 rz 180 deg; joints [-155.421, -81.912, -38.784, 41.861, 38.558, -35.018]
  MoveL 503 to (240.69, 49.94, 22.22) mm, rotated rx -180 ry 0 rz 180 deg; joints [-155.421, -81.912, -38.784, 41.861, 38.558, -35.018]
  Call Extruder(429.95564)
  MoveL 504 to (240.74, 50.24, 22.22) mm, rotated rx 180 ry 0 rz 180 deg; joints [-155.396, -81.937, -38.728, 41.919, 38.55, -35.076]
  MoveL 505 to (240.74, 50.24, 22.22) mm, rotated rx 180 ry 0 rz 180 deg; joints [-155.396, -81.937, -38.728, 41.919, 38.55, -35.076]
  Call Extruder(430.28392)
  MoveL 506 to (240.78, 50.55, 22.23) mm, rotated rx 180 ry 0 rz 180 deg; joints [-155.371, -81.962, -38.673, 41.977, 38.542, -35.134]
  MoveL 507 to (240.78, 50.55, 22.23) mm, rotated rx 180 ry 0 rz 180 deg; joints [-155.371, -81.962, -38.673, 41.977, 38.542, -35.134]
  Call Extruder(430.61048)
  MoveL 508 to (240.83, 50.86, 22.22) mm, rotated rx 180 ry 0 rz 180 deg; joints [-155.346, -81.987, -38.618, 42.036, 38.534, -35.192]
  MoveL 509 to (240.83, 50.86, 22.22) mm, rotated rx 180 ry 0 rz 180 deg; joints [-155.346, -81.987, -38.618, 42.036, 38.534, -35.192]
  Call Extruder(430.97758)
  MoveL 510 to (240.88, 51.2, 22.23) mm, rotated rx 180 ry 0 rz 180 deg; joints [-155.317, -82.015, -38.557, 42.101, 38.526, -35.257]
  MoveL 511 to (240.88, 51.2, 22.23) mm, rotated rx 180 ry 0 rz 180 deg; joints [-155.317, -82.015, -38.557, 42.101, 38.526, -35.257]
  Call Extruder(431.38502)
  MoveL 512 to (240.93, 51.59, 22.22) mm, rotated rx 180 ry 0 rz -180 deg; joints [-155.285, -82.045, -38.491, 42.174, 38.518, -35.329]
  MoveL 513 to (240.93, 51.59, 22.22) mm, rotated rx 180 ry 0 rz -180 deg; joints [-155.285, -82.045, -38.491, 42.174, 38.518, -35.329]
  Call Extruder(431.79041)
  MoveL 514 to (240.97, 51.98, 22.22) mm, rotated rx 180 ry 0 rz 180 deg; joints [-155.252, -82.075, -38.426, 42.246, 38.51, -35.4]
  MoveL 515 to (240.97, 51.98, 22.22) mm, rotated rx 180 ry 0 rz 180 deg; joints [-155.252, -82.075, -38.426, 42.246, 38.51, -35.4]
  Call Extruder(432.19375)
  MoveL 516 to (241.02, 52.36, 22.23) mm, rotated rx -180 ry 0 rz -180 deg; joints [-155.22, -82.105, -38.359, 42.319, 38.503, -35.472]
  MoveL 517 to (241.02, 52.36, 22.23) mm, rotated rx -180 ry 0 rz -180 deg; joints [-155.22, -82.105, -38.359, 42.319, 38.503, -35.472]
  Call Extruder(432.59504)
  MoveL 518 to (241.06, 52.75, 22.23) mm, rotated rx -180 ry 0 rz 180 deg; joints [-155.188, -82.135, -38.293, 42.391, 38.495, -35.544]
  MoveL 519 to (241.06, 52.75, 22.23) mm, rotated rx -180 ry 0 rz 180 deg; joints [-155.188, -82.135, -38.293, 42.391, 38.495, -35.544]
  Call Extruder(433.20001)
  MoveL 520 to (241.11, 53.34, 22.23) mm, rotated rx 180 ry 0 rz 180 deg; joints [-155.138, -82.178, -38.199, 42.5, 38.486, -35.651]
  MoveL 521 to (241.11, 53.34, 22.23) mm, rotated rx 180 ry 0 rz 180 deg; joints [-155.138, -82.178, -38.199, 42.5, 38.486, -35.651]
  Call Extruder(433.80182)
  MoveL 522 to (241.16, 53.93, 22.23) mm, rotated rx -180 ry 0 rz 180 deg; joints [-155.088, -82.221, -38.105, 42.609, 38.478, -35.758]
  MoveL 523 to (241.16, 53.93, 22.23) mm, rotated rx -180 ry 0 rz 180 deg; joints [-155.088, -82.221, -38.105, 42.609, 38.478, -35.758]
  Call Extruder(434.40048)
  MoveL 524 to (241.2, 54.52, 22.23) mm, rotated rx -180 ry 0 rz -180 deg; joints [-155.038, -82.265, -38.01, 42.718, 38.469, -35.865]
  MoveL 525 to (241.2, 54.52, 22.23) mm, rotated rx -180 ry 0 rz -180 deg; joints [-155.038, -82.265, -38.01, 42.718, 38.469, -35.865]
  Call Extruder(435.57226)
  MoveL 526 to (241.25, 55.68, 22.22) mm, rotated rx -180 ry 0 rz -180 deg; joints [-154.938, -82.344, -37.835, 42.93, 38.458, -36.07]
  MoveL 527 to (241.25, 55.68, 22.22) mm, rotated rx -180 ry 0 rz -180 deg; joints [-154.938, -82.344, -37.835, 42.93, 38.458, -36.07]
  Call Extruder(437.02987)
  MoveL 528 to (241.29, 57.14, 22.23) mm, rotated rx 180 ry 0 rz 180 deg; joints [-154.812, -82.442, -37.621, 43.193, 38.448, -36.326]
  Call Extruder(522.92352)
  MoveL 529 to (241.29, 142.86, 22.22) mm, rotated rx 180 ry 0 rz 180 deg; joints [-147.778, -90.02, -21.56, 59.734, 38.123, -53.432]
  Call Extruder(523.79834)
  MoveL 530 to (241.27, 143.73, 22.22) mm, rotated rx 180 ry 0 rz 180 deg; joints [-147.711, -90.125, -21.344, 59.922, 38.121, -53.64]
  MoveL 531 to (241.27, 143.73, 22.22) mm, rotated rx 180 ry 0 rz 180 deg; joints [-147.711, -90.125, -21.344, 59.922, 38.121, -53.64]
  Call Extruder(524.97012)
  MoveL 532 to (241.23, 144.9, 22.23) mm, rotated rx 180 ry 0 rz 180 deg; joints [-147.62, -90.262, -21.062, 60.169, 38.122, -53.912]
  MoveL 533 to (241.23, 144.9, 22.23) mm, rotated rx 180 ry 0 rz 180 deg; joints [-147.62, -90.262, -21.062, 60.169, 38.122, -53.912]
  Call Extruder(525.85826)
  MoveL 534 to (241.18, 145.77, 22.23) mm, rotated rx 180 ry 0 rz 180 deg; joints [-147.551, -90.363, -20.852, 60.354, 38.124, -54.115]
  MoveL 535 to (241.18, 145.77, 22.23) mm, rotated rx 180 ry 0 rz 180 deg; joints [-147.551, -90.363, -20.852, 60.354, 38.124, -54.115]
  Call Extruder(526.46008)
  MoveL 536 to (241.13, 146.36, 22.23) mm, rotated rx -180 ry 0 rz -180 deg; joints [-147.504, -90.429, -20.717, 60.476, 38.128, -54.248]
  MoveL 537 to (241.13, 146.36, 22.23) mm, rotated rx -180 ry 0 rz -180 deg; joints [-147.504, -90.429, -20.717, 60.476, 38.128, -54.248]
  Call Extruder(527.06505)
  MoveL 538 to (241.09, 146.95, 22.22) mm, rotated rx -180 ry 0 rz -180 deg; joints [-147.457, -90.496, -20.58, 60.598, 38.132, -54.382]
  MoveL 539 to (241.09, 146.95, 22.22) mm, rotated rx -180 ry 0 rz -180 deg; joints [-147.457, -90.496, -20.58, 60.598, 38.132, -54.382]
  Call Extruder(527.56965)
  MoveL 540 to (241.04, 147.44, 22.22) mm, rotated rx 180 ry 0 rz 180 deg; joints [-147.417, -90.549, -20.469, 60.698, 38.136, -54.491]
  MoveL 541 to (241.04, 147.44, 22.22) mm, rotated rx 180 ry 0 rz 180 deg; joints [-147.417, -90.549, -20.469, 60.698, 38.136, -54.491]
  Call Extruder(527.97299)
  MoveL 542 to (240.99, 147.83, 22.23) mm, rotated rx -180 ry 0 rz -180 deg; joints [-147.386, -90.59, -20.385, 60.776, 38.141, -54.576]
  MoveL 543 to (240.99, 147.83, 22.23) mm, rotated rx -180 ry 0 rz -180 deg; joints [-147.386, -90.59, -20.385, 60.776, 38.141, -54.576]
  Call Extruder(528.37839)
  MoveL 544 to (240.95, 148.22, 22.23) mm, rotated rx 180 ry 0 rz 180 deg; joints [-147.354, -90.631, -20.301, 60.854, 38.145, -54.66]
  MoveL 545 to (240.95, 148.22, 22.23) mm, rotated rx 180 ry 0 rz 180 deg; joints [-147.354, -90.631, -20.301, 60.854, 38.145, -54.66]
  Call Extruder(528.78583)
  MoveL 546 to (240.9, 148.6, 22.23) mm, rotated rx 180 ry 0 rz -180 deg; joints [-147.322, -90.673, -20.216, 60.932, 38.15, -54.745]
  MoveL 547 to (240.9, 148.6, 22.23) mm, rotated rx 180 ry 0 rz -180 deg; joints [-147.322, -90.673, -20.216, 60.932, 38.15, -54.745]
  Call Extruder(529.19532)
  MoveL 548 to (240.86, 148.99, 22.22) mm, rotated rx -180 ry 0 rz 180 deg; joints [-147.291, -90.714, -20.131, 61.01, 38.155, -54.83]
  MoveL 549 to (240.86, 148.99, 22.22) mm, rotated rx -180 ry 0 rz 180 deg; joints [-147.291, -90.714, -20.131, 61.01, 38.155, -54.83]
  Call Extruder(529.52188)
  MoveL 550 to (240.81, 149.3, 22.23) mm, rotated rx -180 ry 0 rz 180 deg; joints [-147.265, -90.744, -20.069, 61.069, 38.16, -54.894]
  MoveL 551 to (240.81, 149.3, 22.23) mm, rotated rx -180 ry 0 rz 180 deg; joints [-147.265, -90.744, -20.069, 61.069, 38.16, -54.894]
  Call Extruder(529.85015)
  MoveL 552 to (240.76, 149.6, 22.23) mm, rotated rx 180 ry 0 rz 180 deg; joints [-147.24, -90.775, -20.007, 61.128, 38.165, -54.958]
  MoveL 553 to (240.76, 149.6, 22.23) mm, rotated rx 180 ry 0 rz 180 deg; joints [-147.24, -90.775, -20.007, 61.128, 38.165, -54.958]
  Call Extruder(530.18015)
  MoveL 554 to (240.71, 149.91, 22.23) mm, rotated rx 180 ry 0 rz 180 deg; joints [-147.214, -90.805, -19.944, 61.188, 38.171, -55.022]
  MoveL 555 to (240.71, 149.91, 22.23) mm, rotated rx 180 ry 0 rz 180 deg; joints [-147.214, -90.805, -19.944, 61.188, 38.171, -55.022]
  Call Extruder(530.51186)
  MoveL 556 to (240.66, 150.21, 22.23) mm, rotated rx 180 ry 0 rz 180 deg; joints [-147.189, -90.836, -19.882, 61.247, 38.176, -55.086]
  MoveL 557 to (240.66, 150.21, 22.23) mm, rotated rx 180 ry 0 rz 180 deg; joints [-147.189, -90.836, -19.882, 61.247, 38.176, -55.086]
  Call Extruder(530.84529)
  MoveL 558 to (240.61, 150.52, 22.23) mm, rotated rx 180 ry 0 rz 180 deg; joints [-147.163, -90.866, -19.819, 61.307, 38.182, -55.15]
  MoveL 559 to (240.61, 150.52, 22.23) mm, rotated rx 180 ry 0 rz 180 deg; joints [-147.163, -90.866, -19.819, 61.307, 38.182, -55.15]
  Call Extruder(531.18045)
  MoveL 560 to (240.56, 150.83, 22.22) mm, rotated rx 180 ry 0 rz -180 deg; joints [-147.138, -90.897, -19.756, 61.366, 38.187, -55.215]
  MoveL 561 to (240.56, 150.83, 22.22) mm, rotated rx 180 ry 0 rz -180 deg; joints [-147.138, -90.897, -19.756, 61.366, 38.187, -55.215]
  Call Extruder(531.45690)
  MoveL 562 to (240.52, 151.07, 22.23) mm, rotated rx -180 ry 0 rz 180 deg; joints [-147.117, -90.92, -19.708, 61.413, 38.193, -55.265]
  MoveL 563 to (240.52, 151.07, 22.23) mm, rotated rx -180 ry 0 rz 180 deg; joints [-147.117, -90.92, -19.708, 61.413, 38.193, -55.265]
  Call Extruder(531.73480)
  MoveL 564 to (240.47, 151.32, 22.22) mm, rotated rx -180 ry 0 rz -180 deg; joints [-147.095, -90.943, -19.661, 61.459, 38.199, -55.314]
  MoveL 565 to (240.47, 151.32, 22.22) mm, rotated rx -180 ry 0 rz -180 deg; joints [-147.095, -90.943, -19.661, 61.459, 38.199, -55.314]
  Call Extruder(532.01414)
  MoveL 566 to (240.42, 151.57, 22.22) mm, rotated rx 180 ry 0 rz 180 deg; joints [-147.074, -90.966, -19.614, 61.506, 38.205, -55.364]
  MoveL 567 to (240.42, 151.57, 22.22) mm, rotated rx 180 ry 0 rz 180 deg; joints [-147.074, -90.966, -19.614, 61.506, 38.205, -55.364]
  Call Extruder(532.29492)
  MoveL 568 to (240.37, 151.82, 22.23) mm, rotated rx -180 ry 0 rz -180 deg; joints [-147.053, -90.99, -19.566, 61.553, 38.21, -55.414]
  MoveL 569 to (240.37, 151.82, 22.23) mm, rotated rx -180 ry 0 rz -180 deg; joints [-147.053, -90.99, -19.566, 61.553, 38.21, -55.414]
  Call Extruder(532.57714)
  MoveL 570 to (240.32, 152.07, 22.22) mm, rotated rx 180 ry 0 rz 180 deg; joints [-147.032, -91.013, -19.519, 61.599, 38.216, -55.464]
  MoveL 571 to (240.32, 152.07, 22.22) mm, rotated rx 180 ry 0 rz 180 deg; joints [-147.032, -91.013, -19.519, 61.599, 38.216, -55.464]
  Call Extruder(532.86081)
  MoveL 572 to (240.27, 152.32, 22.23) mm, rotated rx 180 ry 0 rz 180 deg; joints [-147.011, -91.036, -19.471, 61.646, 38.222, -55.514]
  MoveL 573 to (240.27, 152.32, 22.23) mm, rotated rx 180 ry 0 rz 180 deg; joints [-147.011, -91.036, -19.471, 61.646, 38.222, -55.514]
  Call Extruder(533.14591)
  MoveL 574 to (240.22, 152.57, 22.22) mm, rotated rx 180 ry 0 rz 180 deg; joints [-146.989, -91.059, -19.423, 61.693, 38.228, -55.564]
  MoveL 575 to (240.22, 152.57, 22.22) mm, rotated rx 180 ry 0 rz 180 deg; joints [-146.989, -91.059, -19.423, 61.693, 38.228, -55.564]
  Call Extruder(533.38165)
  MoveL 576 to (240.17, 152.77, 22.23) mm, rotated rx -180 ry 0 rz 180 deg; joints [-146.972, -91.078, -19.385, 61.731, 38.233, -55.604]
  MoveL 577 to (240.17, 152.77, 22.23) mm, rotated rx -180 ry 0 rz 180 deg; joints [-146.972, -91.078, -19.385, 61.731, 38.233, -55.604]
  Call Extruder(533.61845)
  MoveL 578 to (240.13, 152.98, 22.22) mm, rotated rx -180 ry 0 rz -180 deg; joints [-146.954, -91.096, -19.347, 61.768, 38.239, -55.644]
  MoveL 579 to (240.13, 152.98, 22.22) mm, rotated rx -180 ry 0 rz -180 deg; joints [-146.954, -91.096, -19.347, 61.768, 38.239, -55.644]
  Call Extruder(533.85633)
  MoveL 580 to (240.08, 153.18, 22.22) mm, rotated rx 180 ry 0 rz 180 deg; joints [-146.937, -91.115, -19.31, 61.806, 38.244, -55.684]
  MoveL 581 to (240.08, 153.18, 22.22) mm, rotated rx 180 ry 0 rz 180 deg; joints [-146.937, -91.115, -19.31, 61.806, 38.244, -55.684]
  Call Extruder(534.09527)
  MoveL 582 to (240.04, 153.39, 22.23) mm, rotated rx -180 ry 0 rz -180 deg; joints [-146.919, -91.133, -19.271, 61.844, 38.249, -55.725]
  MoveL 583 to (240.04, 153.39, 22.23) mm, rotated rx -180 ry 0 rz -180 deg; joints [-146.919, -91.133, -19.271, 61.844, 38.249, -55.725]
  Call Extruder(534.34924)
  MoveL 584 to (239.98, 153.6, 22.22) mm, rotated rx 180 ry 0 rz 180 deg; joints [-146.9, -91.151, -19.236, 61.881, 38.256, -55.764]
  MoveL 585 to (239.98, 153.6, 22.22) mm, rotated rx 180 ry 0 rz 180 deg; joints [-146.9, -91.151, -19.236, 61.881, 38.256, -55.764]
  Call Extruder(534.61883)
  MoveL 586 to (239.92, 153.82, 22.23) mm, rotated rx 180 ry 0 rz -180 deg; joints [-146.88, -91.167, -19.202, 61.919, 38.265, -55.803]
  MoveL 587 to (239.92, 153.82, 22.23) mm, rotated rx 180 ry 0 rz -180 deg; joints [-146.88, -91.167, -19.202, 61.919, 38.265, -55.803]
  Call Extruder(534.88976)
  MoveL 588 to (239.85, 154.05, 22.23) mm, rotated rx 180 ry 0 rz 180 deg; joints [-146.86, -91.183, -19.169, 61.956, 38.273, -55.842]
  MoveL 589 to (239.85, 154.05, 22.23) mm, rotated rx 180 ry 0 rz 180 deg; joints [-146.86, -91.183, -19.169, 61.956, 38.273, -55.842]
  Call Extruder(535.16202)
  MoveL 590 to (239.78, 154.27, 22.23) mm, rotated rx 180 ry 0 rz -180 deg; joints [-146.84, -91.2, -19.135, 61.994, 38.282, -55.881]
  MoveL 591 to (239.78, 154.27, 22.23) mm, rotated rx 180 ry 0 rz -180 deg; joints [-146.84, -91.2, -19.135, 61.994, 38.282, -55.881]
  Call Extruder(535.43561)
  MoveL 592 to (239.71, 154.49, 22.23) mm, rotated rx 180 ry 0 rz -180 deg; joints [-146.82, -91.217, -19.101, 62.031, 38.29, -55.92]
  MoveL 593 to (239.71, 154.49, 22.23) mm, rotated rx 180 ry 0 rz -180 deg; joints [-146.82, -91.217, -19.101, 62.031, 38.29, -55.92]
  Call Extruder(535.66881)
  MoveL 594 to (239.65, 154.68, 22.22) mm, rotated rx 180 ry 0 rz 180 deg; joints [-146.803, -91.23, -19.074, 62.062, 38.298, -55.951]
  MoveL 595 to (239.65, 154.68, 22.22) mm, rotated rx 180 ry 0 rz 180 deg; joints [-146.803, -91.23, -19.074, 62.062, 38.298, -55.951]
  Call Extruder(535.90306)
  MoveL 596 to (239.59, 154.87, 22.23) mm, rotated rx 180 ry 0 rz 180 deg; joints [-146.785, -91.243, -19.047, 62.093, 38.306, -55.983]
  MoveL 597 to (239.59, 154.87, 22.23) mm, rotated rx 180 ry 0 rz 180 deg; joints [-146.785, -91.243, -19.047, 62.093, 38.306, -55.983]
  Call Extruder(536.13835)
  MoveL 598 to (239.53, 155.06, 22.22) mm, rotated rx -180 ry 0 rz 180 deg; joints [-146.768, -91.256, -19.021, 62.124, 38.314, -56.015]
  MoveL 599 to (239.53, 155.06, 22.22) mm, rotated rx -180 ry 0 rz 180 deg; joints [-146.768, -91.256, -19.021, 62.124, 38.314, -56.015]
  Call Extruder(536.37470)
  MoveL 600 to (239.47, 155.25, 22.22) mm, rotated rx 180 ry 0 rz 180 deg; joints [-146.751, -91.269, -18.994, 62.155, 38.322, -56.047]
  MoveL 601 to (239.47, 155.25, 22.22) mm, rotated rx 180 ry 0 rz 180 deg; joints [-146.751, -91.269, -18.994, 62.155, 38.322, -56.047]
  Call Extruder(536.61210)
  MoveL 602 to (239.41, 155.44, 22.23) mm, rotated rx 180 ry 0 rz 180 deg; joints [-146.734, -91.282, -18.967, 62.185, 38.329, -56.078]
  MoveL 603 to (239.41, 155.44, 22.23) mm, rotated rx 180 ry 0 rz 180 deg; joints [-146.734, -91.282, -18.967, 62.185, 38.329, -56.078]
  Call Extruder(536.99230)
  MoveL 604 to (239.29, 155.73, 22.23) mm, rotated rx 180 ry 0 rz -180 deg; joints [-146.706, -91.297, -18.936, 62.228, 38.345, -56.12]
  MoveL 605 to (239.29, 155.73, 22.23) mm, rotated rx 180 ry 0 rz -180 deg; joints [-146.706, -91.297, -18.936, 62.228, 38.345, -56.12]
  Call Extruder(537.37429)
  MoveL 606 to (239.17, 156.02, 22.23) mm, rotated rx 180 ry 0 rz -180 deg; joints [-146.678, -91.312, -18.905, 62.27, 38.361, -56.162]
  MoveL 607 to (239.17, 156.02, 22.23) mm, rotated rx 180 ry 0 rz -180 deg; joints [-146.678, -91.312, -18.905, 62.27, 38.361, -56.162]
  Call Extruder(537.73076)
  MoveL 608 to (239.05, 156.29, 22.23) mm, rotated rx 180 ry 0 rz -180 deg; joints [-146.652, -91.326, -18.878, 62.309, 38.376, -56.2]
  MoveL 609 to (239.05, 156.29, 22.23) mm, rotated rx 180 ry 0 rz -180 deg; joints [-146.652, -91.326, -18.878, 62.309, 38.376, -56.2]
  Call Extruder(538.06143)
  MoveL 610 to (238.94, 156.54, 22.23) mm, rotated rx 180 ry 0 rz 180 deg; joints [-146.628, -91.338, -18.853, 62.345, 38.39, -56.235]
  MoveL 611 to (238.94, 156.54, 22.23) mm, rotated rx 180 ry 0 rz 180 deg; joints [-146.628, -91.338, -18.853, 62.345, 38.39, -56.235]
  Call Extruder(538.39353)
  MoveL 612 to (238.84, 156.79, 22.22) mm, rotated rx 180 ry 0 rz 180 deg; joints [-146.604, -91.35, -18.828, 62.381, 38.404, -56.27]
  MoveL 613 to (238.84, 156.79, 22.22) mm, rotated rx 180 ry 0 rz 180 deg; joints [-146.604, -91.35, -18.828, 62.381, 38.404, -56.27]
  Call Extruder(538.82540)
  MoveL 614 to (238.66, 157.09, 22.22) mm, rotated rx -180 ry 0 rz 180 deg; joints [-146.573, -91.355, -18.817, 62.415, 38.428, -56.3]
  MoveL 615 to (238.66, 157.09, 22.22) mm, rotated rx -180 ry 0 rz 180 deg; joints [-146.573, -91.355, -18.817, 62.415, 38.428, -56.3]
  Call Extruder(539.25912)
  MoveL 616 to (238.49, 157.4, 22.22) mm, rotated rx 180 ry 0 rz 180 deg; joints [-146.542, -91.361, -18.806, 62.449, 38.451, -56.33]
  MoveL 617 to (238.49, 157.4, 22.22) mm, rotated rx 180 ry 0 rz 180 deg; joints [-146.542, -91.361, -18.806, 62.449, 38.451, -56.33]
  Call Extruder(539.69468)
  MoveL 618 to (238.31, 157.7, 22.23) mm, rotated rx 180 ry 0 rz -180 deg; joints [-146.51, -91.366, -18.795, 62.484, 38.475, -56.36]
  MoveL 619 to (238.31, 157.7, 22.23) mm, rotated rx 180 ry 0 rz -180 deg; joints [-146.51, -91.366, -18.795, 62.484, 38.475, -56.36]
  Call Extruder(540.13207)
  MoveL 620 to (238.14, 158.01, 22.22) mm, rotated rx -180 ry 0 rz 180 deg; joints [-146.479, -91.371, -18.784, 62.518, 38.498, -56.39]
  MoveL 621 to (238.14, 158.01, 22.22) mm, rotated rx -180 ry 0 rz 180 deg; joints [-146.479, -91.371, -18.784, 62.518, 38.498, -56.39]
  Call Extruder(540.50882)
  MoveL 622 to (237.96, 158.25, 22.22) mm, rotated rx -180 ry 0 rz -180 deg; joints [-146.452, -91.368, -18.79, 62.538, 38.522, -56.405]
  MoveL 623 to (237.96, 158.25, 22.22) mm, rotated rx -180 ry 0 rz -180 deg; joints [-146.452, -91.368, -18.79, 62.538, 38.522, -56.405]
  Call Extruder(541.20873)
  MoveL 624 to (237.63, 158.7, 22.22) mm, rotated rx -180 ry 0 rz -180 deg; joints [-146.402, -91.362, -18.803, 62.576, 38.567, -56.43]
  MoveL 625 to (237.63, 158.7, 22.22) mm, rotated rx -180 ry 0 rz -180 deg; joints [-146.402, -91.362, -18.803, 62.576, 38.567, -56.43]
  Call Extruder(541.91145)
  MoveL 626 to (237.3, 159.15, 22.23) mm, rotated rx 180 ry 0 rz 180 deg; joints [-146.352, -91.357, -18.814, 62.613, 38.611, -56.456]
  Call Extruder(543.65031)
  MoveL 627 to (236.39, 160.19, 22.22) mm, rotated rx -180 ry 0 rz 180 deg; joints [-146.229, -91.31, -18.909, 62.668, 38.736, -56.472]
  Call Extruder(545.38913)
  MoveL 628 to (235.35, 161.1, 22.23) mm, rotated rx 180 ry 0 rz 180 deg; joints [-146.109, -91.221, -19.092, 62.67, 38.878, -56.422]
  Call Extruder(545.74051)
  MoveL 629 to (235.13, 161.27, 22.22) mm, rotated rx 180 ry 0 rz 180 deg; joints [-146.086, -91.197, -19.141, 62.663, 38.91, -56.402]
  MoveL 630 to (235.13, 161.27, 22.22) mm, rotated rx 180 ry 0 rz 180 deg; joints [-146.086, -91.197, -19.141, 62.663, 38.91, -56.402]
  Call Extruder(546.44047)
  MoveL 631 to (234.68, 161.59, 22.23) mm, rotated rx 180 ry 0 rz 180 deg; joints [-146.039, -91.149, -19.24, 62.65, 38.972, -56.364]
  MoveL 632 to (234.68, 161.59, 22.23) mm, rotated rx 180 ry 0 rz 180 deg; joints [-146.039, -91.149, -19.24, 62.65, 38.972, -56.364]
  Call Extruder(547.13763)
  MoveL 633 to (234.22, 161.92, 22.23) mm, rotated rx 180 ry 0 rz 180 deg; joints [-145.992, -91.101, -19.337, 62.636, 39.034, -56.325]
  MoveL 634 to (234.22, 161.92, 22.23) mm, rotated rx 180 ry 0 rz 180 deg; joints [-145.992, -91.101, -19.337, 62.636, 39.034, -56.325]
  Call Extruder(547.38444)
  MoveL 635 to (234.05, 162.02, 22.23) mm, rotated rx 180 ry 0 rz 180 deg; joints [-145.976, -91.08, -19.381, 62.626, 39.058, -56.304]
  MoveL 636 to (234.05, 162.02, 22.23) mm, rotated rx 180 ry 0 rz 180 deg; joints [-145.976, -91.08, -19.381, 62.626, 39.058, -56.304]
  Call Extruder(547.82000)
  MoveL 637 to (233.75, 162.2, 22.23) mm, rotated rx 180 ry 0 rz 180 deg; joints [-145.947, -91.042, -19.459, 62.607, 39.1, -56.267]
  MoveL 638 to (233.75, 162.2, 22.23) mm, rotated rx 180 ry 0 rz 180 deg; joints [-145.947, -91.042, -19.459, 62.607, 39.1, -56.267]
  Call Extruder(548.25372)
  MoveL 639 to (233.45, 162.37, 22.22) mm, rotated rx 180 ry 0 rz -180 deg; joints [-145.919, -91.003, -19.538, 62.588, 39.142, -56.23]
  MoveL 640 to (233.45, 162.37, 22.22) mm, rotated rx 180 ry 0 rz -180 deg; joints [-145.919, -91.003, -19.538, 62.588, 39.142, -56.23]
  Call Extruder(548.68559)
  MoveL 641 to (233.14, 162.55, 22.22) mm, rotated rx -180 ry 0 rz -180 deg; joints [-145.891, -90.965, -19.616, 62.57, 39.184, -56.194]
  MoveL 642 to (233.14, 162.55, 22.22) mm, rotated rx -180 ry 0 rz -180 deg; joints [-145.891, -90.965, -19.616, 62.57, 39.184, -56.194]
  Call Extruder(549.06597)
  MoveL 643 to (232.87, 162.69, 22.22) mm, rotated rx 180 ry 0 rz 180 deg; joints [-145.866, -90.928, -19.691, 62.549, 39.222, -56.156]
  MoveL 644 to (232.87, 162.69, 22.22) mm, rotated rx 180 ry 0 rz 180 deg; joints [-145.866, -90.928, -19.691, 62.549, 39.222, -56.156]
  Call Extruder(549.39656)
  MoveL 645 to (232.62, 162.8, 22.23) mm, rotated rx 180 ry 0 rz 180 deg; joints [-145.845, -90.892, -19.765, 62.526, 39.256, -56.117]
  MoveL 646 to (232.62, 162.8, 22.23) mm, rotated rx 180 ry 0 rz 180 deg; joints [-145.845, -90.892, -19.765, 62.526, 39.256, -56.117]
  Call Extruder(549.72573)
  MoveL 647 to (232.37, 162.91, 22.23) mm, rotated rx 180 ry 0 rz 180 deg; joints [-145.825, -90.857, -19.839, 62.503, 39.291, -56.078]
  MoveL 648 to (232.37, 162.91, 22.23) mm, rotated rx 180 ry 0 rz 180 deg; joints [-145.825, -90.857, -19.839, 62.503, 39.291, -56.078]
  Call Extruder(550.10778)
  MoveL 649 to (232.07, 163.02, 22.23) mm, rotated rx 180 ry 0 rz -180 deg; joints [-145.801, -90.814, -19.926, 62.476, 39.331, -56.032]
  MoveL 650 to (232.07, 163.02, 22.23) mm, rotated rx 180 ry 0 rz -180 deg; joints [-145.801, -90.814, -19.926, 62.476, 39.331, -56.032]
  Call Extruder(550.48803)
  MoveL 651 to (231.78, 163.15, 22.23) mm, rotated rx 180 ry 0 rz -180 deg; joints [-145.777, -90.772, -20.013, 62.448, 39.372, -55.985]
  MoveL 652 to (231.78, 163.15, 22.23) mm, rotated rx 180 ry 0 rz -180 deg; joints [-145.777, -90.772, -20.013, 62.448, 39.372, -55.985]
  Call Extruder(550.79572)
  MoveL 653 to (231.54, 163.24, 22.22) mm, rotated rx 180 ry 0 rz 180 deg; joints [-145.759, -90.736, -20.087, 62.424, 39.405, -55.946]
  MoveL 654 to (231.54, 163.24, 22.22) mm, rotated rx 180 ry 0 rz 180 deg; joints [-145.759, -90.736, -20.087, 62.424, 39.405, -55.946]
  Call Extruder(551.03204)
  MoveL 655 to (231.35, 163.3, 22.23) mm, rotated rx -180 ry 0 rz 180 deg; joints [-145.744, -90.706, -20.147, 62.403, 39.431, -55.912]
  MoveL 656 to (231.35, 163.3, 22.23) mm, rotated rx -180 ry 0 rz 180 deg; joints [-145.744, -90.706, -20.147, 62.403, 39.431, -55.912]
  Call Extruder(551.26731)
